(* Logix 5000 project; controller DispersionPlc vendor 1 type 14 code 108 rev 34.11; software revision 34.01; part 3 of 22 *)
(* tags used below, declared in another part *)
   Control_Rm_tags : DINT;
   Dev : REAL[10];
   DevAlarms : DINT;
   DevTimer : TIMER[10];
   Dispersion_to_Main : DINT;
   Dispersion_to_Main2 : DINT;
   Dispersion_to_SIL2 : DINT;
   Dispersion_to_SIL2_Analog : REAL[24];
   GenPurp : AStd_GeneralPurp;
   PLCStatus : AStd_PLCStatus;
   SP : REAL;

   T4301_AIR_PURGE : ALIAS FOR Local:6:O.Data.4;
   T4301_AIR_PURGE_AUTO : BOOL := 1;
   T4301_AIR_PURGE_REQUEST : BOOL;
   T4301_COOLING_NOT_PURGED : BOOL;
   T4301_COOLING_OCCURED : BOOL;
   T4301_Cooling_On : BOOL;
   T4301_COOLING_OPERATION : BOOL;
   T4301_Cooling_Reset_TMR : TIMER := (PRE := 500);
   T4301_COOLING_TEMP : DINT := 72;
   T4301_COOLING_VALVE : ALIAS FOR Local:6:O.Data.3;
   T4301_COOLING_VALVE_HMI : BOOL;
   T4301_DISCHARGE : BOOL;
   T4301_DISCHARGE_VALVE : AB:1769_DI16:I:0;
   T4301_Heating_On : BOOL;
   T4301_HEATING_OPERATION : BOOL;
   T4301_HMI_Cooling : BOOL;
   T4301_HMI_Heating : BOOL;
   T4301_K : Kettle := (Heating.Value := 78.0, Heating.Setpoint := 100.0, Heating.Error_Val := 115.0, Heating.OUT := 10000.0, Cooling.Value := 78.0, Cooling.Setpoint := 85.0, Cooling.Error_Val := 72.0, Cooling.OUT := 10000.0, Combined.Value := 78.0, Auto_Manual := 1, Cool_Auto_Manual := 1);
   T4301_Manual_AIR_PURGE_REQUEST : BOOL;
   T4301_Mixer : VFD := (TargetDriveSpeed := 100, I_CmdDir := 1, I_ActDir := 1, I_LocalContStat1 := 1, I_LocalContStat2 := 1, I_LocalContStat3 := 1, O_Stop := 1, O_DirBit1 := 1, O_Reff_Sel1 := 1, O_V_CmdReff := 11000.0, SpeedScaleIn := 110.0, SpeedScaleOut := 110.0, MaxOutPut := 100.0, MinOutput := 10.0);
   T4301_Mixer_Enable : DINT;
   T4301_PID_Setpoints : PID[5] := ([1].SP := 100.0, [1].KP := 325.0, [1].KI := 0.02, [2].KP := 9.0, [2].KI := 8.0, [2].KD := 7.0, [3].KP := 8.0, [3].KI := 0.2, [4].KP := 6.0, [4].KI := 5.0, [4].KD := 4.0);
   T4301_Pids_On : BOOL;
   T4301_Post_PurgeTm : DINT := 20000;
   T4301_Pre_PurgeTm : DINT := 2000;
   T4301_PrePurgeTMR : TIMER := (PRE := 2000);
   T4301_Process_Alarm_Setpoints : Alarm_SPT := (HIHI := 340.0, HI := 320.0);
   T4301_Purge_Complete : BOOL := 1;
   T4301_Request_Cooling : BOOL;
   T4301_Request_Cooling_Tmr : TIMER[5] := ([0].PRE := 30000, [1].PRE := 30000, [2].PRE := 500, [3].PRE := 8000, [4].PRE := 500, [4].ACC := 515, [4].EN := 1, [4].DN := 1);
   T4301_Request_Cooling_Tmr1 : TIMER := (PRE := 1000);
   T4301_Request_Heating : BOOL;
   T4301_Request_Heating_Hold : BOOL;
   T4301_Request_Heating_Tmr : TIMER[5] := ([0].PRE := 5000, [4].PRE := 5000, [4].ACC := 5006);
   T4301_Stop_Pids : BOOL;
   T4301_T4302_Xfer_In_Enable_Ctrl : BOOL := 1;
   T4301_Temp_Feed_Alarm : DINT := 310;
   T4301_Z1_HEAT_VALVE : ALIAS FOR Local:6:O.Data.0;
   T4301_Z2_HEAT_VALVE : ALIAS FOR Local:6:O.Data.1;
   T4301_Z3_HEAT_VALVE : ALIAS FOR Local:6:O.Data.2;
   T4301ons2 : DINT := 386;
   T4301PID_I : REAL;
   T4301Purge : Seq64 := (Val := 1, Tmr[3].PRE := 4000, Tmr[5].PRE := 20000, Sq.Step[1] := 1);
   T4302_AIR_PURGE : ALIAS FOR Local:6:O.Data.13;
   T4302_AIR_PURGE_AUTO : BOOL := 1;
   T4302_AIR_PURGE_REQUEST : BOOL;
   T4302_Cooling_No_Heat : TIMER := (PRE := 200000);
   T4302_COOLING_NOT_PURGED : BOOL;
   T4302_COOLING_OCCURED : BOOL;
   T4302_Cooling_On : BOOL := 1;
   T4302_COOLING_OPERATION : BOOL := 1;
   T4302_Cooling_Pressure : DINT;
   T4302_Cooling_Pressure_SPT : DINT := 50;
   T4302_COOLING_TEMP : DINT := 2192;
   T4302_COOLING_VALVE : ALIAS FOR Local:6:O.Data.10;
   T4302_COOLING_VALVE_HMI : BOOL;
   T4302_DISCHARGE : BOOL;
   T4302_Heating_On : BOOL;
   T4302_HEATING_OPERATION : BOOL;
   T4302_HMI_Cooling : BOOL;
   T4302_HMI_Heating : BOOL;
   T4302_K : Kettle := (Heating.Value := 65.0, Heating.Setpoint := 150.0, Heating.Error_Val := 95.0, Heating.OUT := 5000.0, Cooling.Value := 65.0, Cooling.Setpoint := 180.0, Combined.Value := 65.0, Combined.Setpoint := 287.0, Auto_Manual := 1, ValveOutput := 2, Cool_Auto_Manual := 1);
   t4302_Line_pressure_High : BOOL;
   t4302_Line_pressure_Hightmr : TIMER := (PRE := 20000);
   T4302_Manual_AIR_PURGE_REQUEST : BOOL;
   T4302_Mixer : VFD := (TargetDriveSpeed := 100, I_DatalinkA2_Fb := 223.0, O_DirBit1 := 1, O_Reff_Sel1 := 1, O_V_CmdReff := 11000.0, SpeedScaleIn := 110.0, SpeedScaleOut := 110.0, MaxOutPut := 100.0, MinOutput := 10.0);
   T4302_Phase_S52_Transfer : AStd_PLI := (IdleS := 1, CurrentStateCodeS := 1, PreventStartS := 2, AlarmS := 2, StepNo := 1, StepBit := 2, PreventStartInhibitC := 3, AlarmInhibitC := 3, IntSafDisp := 2);
   T4302_Phase_S52_Transfer_AOI : AStd_PLI_AOI := (PreventStartS := 1, AlmS := 1, StepNo := 1, cfgAutoReset := 1);
   T4302_Phase_TT_Transfer : AStd_PLI := (IdleS := 1, CurrentStateCodeS := 1, PreventStartS := 2, AlarmS := 2, StepNo := 1, StepBit := 2, RealParameters[0] := 44000.0, PreventStartInhibitC := 7, AlarmInhibitC := 3, IntSafDisp := 2);
   T4302_Phase_TT_Transfer_AOI : AStd_PLI_AOI := (PreventStartS := 1, AlmS := 1, StepNo := 1, cfgAutoReset := 1);
   T4302_PhaseAgitation : AStd_PLI := (IdleS := 1, CurrentStateCodeS := 1, StepNo := 1, StepBit := 2, DINTParameters[0] := 32, DINTParameters[1] := 8500, PreventStartInhibitC := 3, AlarmInhibitC := 3);
   T4302_PhaseAgitation_AOI : AStd_PLI_AOI := (StepNo := 1, cfgAutoReset := 1);
   T4302_PhaseTempControl : AStd_PLI := (IdleS := 1, CurrentStateCodeS := 1, StepNo := 1, StepBit := 2, RealParameters[0] := 65.0, RealParameters[1] := 64.0, RealParameters[3] := 50.0, RealParameters[4] := 113.0, RealParameters[5] := 50.0, RealParameters[10] := 5000.0, RealParameters[19] := 70.0, DINTParameters[0] := 5, DINTParameters[19] := 80, PreventStartInhibitC := 15, AlarmInhibitC := 15);
   T4302_PhaseTempControl_AOI : AStd_PLI_AOI := (StepNo := 1, cfgAutoReset := 1);
   T4302_PID_Setpoints : PID[5] := ([1].SP := 5.0, [1].KP := 150.0, [1].KI := 0.01, [2].KP := 9.0, [2].KI := 8.0, [2].KD := 7.0, [3].SP := 100.0, [3].KP := 8.0, [3].KI := 0.2, [4].KP := 6.0, [4].KI := 5.0, [4].KD := 4.0);
   T4302_Pids_On : BOOL := 1;
   T4302_Post_PurgeTm : DINT := 20000;
   T4302_Pre_PurgeTm : DINT := 2000;
   T4302_PrePurgeTMR : TIMER := (PRE := 2000);
   T4302_Process_Alarm_Setpoints : Alarm_SPT := (HIHI := 340.0, HI := 320.0);
   T4302_Purge_Complete : BOOL := 1;
   T4302_RampControl : BOOL;
   T4302_RampControl_ONS : BOOL;
   T4302_RampControl_ONS_2 : BOOL;
   T4302_RampControlTOn : TIMER := (PRE := 600000);
   T4302_Request_Cooling : BOOL;
   T4302_Request_Cooling_Tmr : TIMER[5] := ([0].PRE := 20000, [1].PRE := 20000, [2].PRE := 500, [3].PRE := 8000, [4].PRE := 500, [4].ACC := 506, [4].EN := 1, [4].DN := 1);
   T4302_Request_Heating : BOOL;
   T4302_Request_Heating_Hold : BOOL;
   T4302_Request_Heating_Tmr : TIMER[5] := ([0].PRE := 1000, [4].PRE := 1000, [4].ACC := 1000);
   T4302_Stop_Pids : BOOL;
   T4302_Temp_Feed_Alarm : DINT := 310;
   T4302_TransferStarted : BOOL;
   T4302_Z1_HEAT_VALVE : ALIAS FOR Local:6:O.Data.9;
   T4302_Z2_HEAT_VALVE : ALIAS FOR Local:6:O.Data.8;
   T4302_Z3_HEAT_VALVE : ALIAS FOR Local:6:O.Data.11;
   T4302ons2 : DINT := 258;
   T4302Ons3 : BOOL := 1;
   T4302ons4 : BOOL;
   T4302Purge : Seq64 := (Val := 1, Tmr[3].PRE := 4000, Tmr[5].PRE := 2000, Sq.Step[1] := 1);
   T4302TruckTransferCompletePB : BOOL;
   T430_Z3_HEAT_VALVE : ALIAS FOR Local:6:O.Data.11;
   T47_Amount_Per_Count : REAL;
   T47_Charge_Remaining : REAL;
   T47_Flow_Rate : REAL;
   T47_Flow_Raw : DINT;
   T47_Flow_Raw_Adjusted : REAL;
   T47_Flow_Scale_Factor : REAL;
   T47_Last_Charge : REAL;
   T47_Manual_Start : BOOL;
   T47_Max_Flow : REAL;
   T47_Pump_Manual_Run : BOOL;
   T47_Pump_Off : BOOL;
   T47_Pump_Run : BOOL;
   T47_Transfer : BOOL;
   T47_transfer_amount : REAL;
   T47PumpTmr : TIMER;
   T51_Tank_Max_Lbs : REAL := 75000.0;
   T52_Mixer : VFD := (TargetDriveSpeed := 30, I_Ready := 1, I_CmdDir := 1, I_ActDir := 1, I_LocalContStat1 := 1, I_LocalContStat2 := 1, I_LocalContStat3 := 1, O_V_CmdReff := 4530.0, SpeedScaleIn := 151.0, SpeedScaleOut := 151.0, MaxOutPut := 100.0, MinOutput := 10.0);
   T52_Mixer_STOP : TIMER := (PRE := 200, ACC := 202, EN := 1, DN := 1);
   T52_Ons : BOOL[32] := ([20] := 1);
   T52_Selected_For_Pumping : BOOL;
   T52_Tank_Max_Lbs : REAL := 108286.0;
   T52_WARN_BYPASS : BOOL;
   T53_Mixer : VFD := (TargetDriveSpeed := 30, I_Ready := 1, I_CmdDir := 1, I_ActDir := 1, I_LocalContStat1 := 1, I_LocalContStat2 := 1, I_LocalContStat3 := 1, O_V_CmdReff := 4530.0, SpeedScaleIn := 151.0, SpeedScaleOut := 151.0, MaxOutPut := 100.0, MinOutput := 10.0);
   T53_Mixer_STOP : TIMER := (PRE := 200, ACC := 201, EN := 1, DN := 1);
   T53_Ons : BOOL[32];
   T53_Selected_For_Pumping : BOOL := 1;
   T53_Tank_Max_Lbs : REAL := 108286.0;
   T53_WARN_BYPASS : BOOL;
   T_4301_Temp_Holding : REAL := 78.06781;
   T_4301_Temp_Samples : REAL := 1000.0;
   T_4302_Temp_Holding : REAL := 66.95962;
   T_4302_Temp_Samples : REAL := 1000.0;
   T_4302_Temp_Smoothed : REAL := 66.95962;
   TA_4303 : ALIAS FOR Local:7:O.Data.13;
   TAH_4304 : ALIAS FOR Local:7:O.Data.12;
   Tank : Udt_Tank[64];
   tank1 : DINT;
   Tank47_Level : INT;
   Tank47_LevelHiHiAlarm : BOOL;
   Tank_Destination : DINT;
   Tank_Destination_ONS : BOOL;
   Tank_Destination_ONS1 : BOOL;
   Tank_Link_Enable : BOOL := 1;
   Tank_Link_Enable_ONS : BOOL;
   Tank_Link_Enable_ONS1 : BOOL;
   Tank_Link_ONS : BOOL[32];
   Tank_Linked : BOOL := 1;
   Task_OLD_Permissive : BOOL[64];
   Task_Permissive : DINT[2] := ([0] := 4, [1] := 4);
   TC_4305_1 : AStd_PIDInterface := (AutoS := 1, SPC := 65.0, PGainC := 1.0, IGainC := 0.33, DGainC := 0.22, PGainS := 1.0, IGainS := 0.33, DGainS := 0.22, SPS := 65.0, PVS := 76.673004, Perm.IntlkS := 1, Perm.SafeS := 1);
   TC_4305_1_AOI : AStd_PIDInterface_AOI := (SP := 65.0, PV := 76.642, cfgPVMaxEU := 350.0);
   TC_4305_1_PID : PID_ENHANCED := (PV := 76.673004, PVEUMax := 350.0, SPProg := 65.0, SPOper := 65.0, SPHLimit := 350.0, RatioProg := 1.0, RatioOper := 1.0, RatioHLimit := 1.0, RatioLLimit := 1.0, CVEUMax := 100.0, CVHLimit := 100.0, DependIndepend := 1, PGain := 1.0, IGain := 0.33, DGain := 0.22, PVHHLimit := 350.0, PVHLimit := 350.0, PVLLimit := 0.1, PVLLLimit := 0.1, DevHHLimit := 5.0, DevDeadband := 2.0, ProgProgReq := 1, ProgOverrideReq := 1, RTSTime := 1, SP := 65.0, SPPercent := 18.571428, PVPercent := 21.906572, E := -11.673004, EPercent := -3.335144, InitPrimary := 1, Ratio := 1.0, DevHHAlarm := 1, ProgOper := 1, Override := 1, DeltaT := 0.1);
   TCV_4302_1 : AStd_VlvModulating := (AutoC := 1, AutoS := 1, Perm.IntlkS := 1, Perm.SafeS := 1, Perm.InterlockInhibitC := 3, Scaling.RawMaxS := 10000.0, Scaling.EngMaxS := 100.0);
   TCV_4302_1_AOI : AStd_VlVModulating_AOI := (cfgEUMax := 100.0, cfgRawMax := 10000.0, AutoS := 1);
   TCV_4302_2 : AStd_VlvModulating := (AutoC := 1, AutoS := 1, Perm.IntlkS := 1, Perm.SafeS := 1, AutoPosC[0] := 100.0, AutoPosS := 100.0, Scaling.RawMaxS := 10000.0, Scaling.EngMaxS := 100.0);
   TCV_4302_2_AOI : AStd_VlVModulating_AOI := (cfgEUMax := 100.0, cfgRawMax := 10000.0, AutoS := 1);
   TCV_4302_2_Mode : SINT := 1;
   TCV_4305_1 : AStd_VlvModulating := (AutoC := 1, AutoS := 1, Perm.IntlkS := 1, Perm.SafeS := 1, Perm.InterlockInhibitC := 3, Perm.SafetyInhibitC := 255, Scaling.RawMaxS := 10000.0, Scaling.EngMaxS := 100.0);
   TCV_4305_1_AOI : AStd_VlVModulating_AOI := (cfgEUMax := 100.0, cfgRawMax := 10000.0, AutoS := 1);
   TCV_S47_1 : AStd_AnalogInput := (Raw := 4000.0, Scaled := 644000.0, Scaling.RawMaxS := 100.0, Scaling.EngMinS := 4000.0, Scaling.EngMaxS := 20000.0, High.LatchA := 1, High.DetectS := 1, High.BitS := 1, High.Tmr.PRE := 1000, High.Tmr.ACC := 1003, High.Tmr.EN := 1, High.Tmr.DN := 1, HighHigh.LatchA := 1, HighHigh.DetectS := 1, HighHigh.BitS := 1, HighHigh.Tmr.PRE := 1000, HighHigh.Tmr.ACC := 1003, HighHigh.Tmr.EN := 1, HighHigh.Tmr.DN := 1);
   TCV_S47_1_AOI : AStd_AI_AOI := (InputRaw_I := 4000.0, cfgRawMax := 100.0, cfgEUMin := 4000.0, cfgEUMax := 20000.0, Scaled := 644000.0);
   TCV_S47_1_AutoCommand : REAL;
   TCV_S47_1_AutoManTransition : BOOL;
   TCV_S47_1_AutoManTransitionDelay : TIMER := (PRE := 500);
   TCV_S47_1_AutoPB : BOOL;
   TCV_S47_1_AutoSelected : BOOL;
   TCV_S47_1_Command : REAL;
   TCV_S47_1_ManAutoTransition : BOOL;
   TCV_S47_1_ManAutoTransitionDelay : TIMER := (PRE := 500);
   TCV_S47_1_ManualCommand : DINT;
   TCV_S47_1_ManualPB : BOOL;
   TCV_S47_1_ManualSelected : BOOL;
   TCV_S47_1Output : Analog_Scale := (Analog_Max_In := 100.0, Analog_Min_Out := 4000.0, Analog_Max_Out := 20000.0, Analog_Out := 4000.0);
   TE_4301A : ALIAS FOR Local:8:I.Ch0Data;
   Te_4301A_High : REAL := 420.0;
   TE_4301A_Low : REAL := 20.0;
   Te_4301A_max : REAL;
   TE_4301B : ALIAS FOR Local:8:I.Ch1Data;
   TE_4301C : REAL;
   TE_4301D : ALIAS FOR Local:8:I.Ch3Data;
   TE_4301E : ALIAS FOR Local:8:I.Ch4Data;
   TE_4302A : ALIAS FOR Local:8:I.Ch5Data;
   TE_4302A_High : REAL := 420.0;
   TE_4302A_Low : REAL := 20.0;
   TE_4302B : REAL;
   TE_4302C : ALIAS FOR Local:8:I.Ch2Data;
   TE_4302D : REAL;
   TE_4302E : REAL;
   TE_4303 : ALIAS FOR Local:9:I.Ch4Data;
   TE_4303_01 : REAL := 66.38342;
   TE_4303_High : REAL := 90.0;
   TE_4304 : ALIAS FOR Local:9:I.Ch5Data;
   TE_4304_High : REAL := 95.0;
   TE_4320 : INT := 143;
   TE_4320_High : REAL := 160.0;
   TE_4320_Raw : DINT;
   TE_K400_1 : REAL := 5.0;
   TE_K400_1_HIGH : REAL := 300.0;
   TE_K400_1_LOW : REAL := 50.0;
   TempChange : REAL := 54.0;
   TempDifferenceCooling4301 : DINT := 14;
   TempDifferenceCooling4301TMR : TIMER := (PRE := 600000);
   TempDifferenceCooling4302 : DINT := -115;
   TempDifferenceCooling4302TMR : TIMER := (PRE := 600000);
   test1 : BOOL;
   test3 : BOOL;
   TEST_1 : INT;
   TEST_2 : BOOL;
   test_618 : BOOL := 1;
   TEST_INTERLOCK_K400 : BOOL;
   TEST_INTERLOCK_RESET : DINT;
   TEST_INTERLOCK_T4301 : BOOL;
   TEST_INTERLOCK_T4302 : BOOL;
   test_onsite_512 : BOOL;
   test_onsite_514 : BOOL;
   Test_PID : PID_ENHANCED := (PVEUMax := 100.0, SPHLimit := 100.0, RatioProg := 1.0, RatioOper := 1.0, RatioHLimit := 1.0, RatioLLimit := 1.0, CVEUMax := 100.0, CVHLimit := 100.0, PVEDerivative := 1, RTSTime := 1, InitPrimary := 1, Ratio := 1.0, Manual := 1, DeltaT := 0.1);
   TestBit1 : BOOL;
   TestBit2 : BOOL;
   TestBit3 : BOOL := 1;
   testint : DINT;
   testons : DINT;
   testtmr : TIMER[5] := ([0].PRE := 500, [1].PRE := 500, [1].ACC := 500, [1].EN := 1, [1].DN := 1);
   tete : BOOL;
   tg : BOOL;
   THINONS1 : BOOL;
   THO_MSG : MESSAGE;
        MessageParameters(ServiceCode := 16#0fa2, LocalElement := TO_N12[0], ...)
   THRM_OX_ALM_AUX : ALIAS FOR Local:1:I.Data[1].17;
   TIC_4302_1 : AStd_PIDInterface := (AutoS := 1, SPC := 167.0, PGainC := 5.0, IGainC := 0.1, DGainC := 0.5, PGainS := 5.0, IGainS := 0.1, DGainS := 0.5, SPS := 167.0, PVS := 75.0, Perm.IntlkS := 1, Perm.SafeS := 1);
   TIC_4302_1_AOI : AStd_PIDInterface_AOI := (SP := 167.0, PV := 75.0, cfgPVMaxEU := 400.0);
   TIC_4302_1_PID : PID_ENHANCED := (PV := 75.0, PVEUMax := 400.0, SPProg := 167.0, SPOper := 167.0, SPHLimit := 400.0, RatioProg := 1.0, RatioOper := 1.0, RatioHLimit := 1.0, RatioLLimit := 1.0, CVEUMax := 225.0, CVEUMin := 70.0, CVHLimit := 100.0, PGain := 5.0, IGain := 0.1, DGain := 0.5, PVEDerivative := 1, DevDeadband := 2.0, ProgProgReq := 1, ProgOverrideReq := 1, RTSTime := 1, CVEU := 70.0, SP := 167.0, SPPercent := 41.75, PVPercent := 18.75, E := 92.0, EPercent := 23.0, InitPrimary := 1, Ratio := 1.0, ProgOper := 1, Override := 1, DeltaT := 0.1);
   TIC_4302_4C : AStd_PIDInterface := (AutoS := 1, SPC := 65.0, PGainC := 3.9, IGainC := 0.28, DGainC := 0.125, PGainS := 3.9, IGainS := 0.28, DGainS := 0.125, SPS := 65.0, PVS := 75.991, Perm.IntlkS := 1, Perm.SafeS := 1);
   TIC_4302_4C_AOI : AStd_PIDInterface_AOI := (SP := 65.0, PV := 76.022, cfgPVMinEU := 40.0, cfgPVMaxEU := 350.0);
   TIC_4302_4C_PID : PID_ENHANCED := (PV := 76.022, PVEUMax := 350.0, PVEUMin := 40.0, SPProg := 65.0, SPOper := 65.0, SPHLimit := 350.0, SPLLimit := 40.0, RatioProg := 1.0, RatioOper := 1.0, RatioHLimit := 1.0, RatioLLimit := 1.0, CVEUMax := 100.0, CVHLimit := 100.0, ControlAction := 1, DependIndepend := 1, PGain := 3.9, IGain := 0.28, DGain := 0.125, DevDeadband := 2.0, ProgProgReq := 1, ProgOverrideReq := 1, RTSTime := 1, SP := 65.0, SPPercent := 8.064516, PVPercent := 11.609999, E := 10.990997, EPercent := 3.5454826, InitPrimary := 1, Ratio := 1.0, ProgOper := 1, Override := 1, DeltaT := 0.1);
   TIC_4302_4H : AStd_PIDInterface := (AutoS := 1, SPC := 65.0, PGainC := 4.8, IGainC := 0.31, DGainC := 0.19, PGainS := 4.8, IGainS := 0.31, DGainS := 0.19, SPS := 65.0, PVS := 76.022, Perm.IntlkS := 1, Perm.SafeS := 1);
   TIC_4302_4H_AOI : AStd_PIDInterface_AOI := (SP := 65.0, PV := 76.022, cfgPVMinEU := 40.0, cfgPVMaxEU := 350.0);
   TIC_4302_4H_PID : PID_ENHANCED := (PV := 76.022, PVEUMax := 350.0, PVEUMin := 40.0, SPProg := 65.0, SPOper := 65.0, SPHLimit := 350.0, SPLLimit := 40.0, RatioProg := 1.0, RatioOper := 1.0, RatioHLimit := 1.0, RatioLLimit := 1.0, CVEUMax := 100.0, CVHLimit := 80.0, DependIndepend := 1, PGain := 4.8, IGain := 0.31, DGain := 0.19, DevDeadband := 2.0, ProgProgReq := 1, ProgOverrideReq := 1, RTSTime := 1, SP := 65.0, SPPercent := 8.064516, PVPercent := 11.620001, E := -11.022003, EPercent := -3.5554848, InitPrimary := 1, Ratio := 1.0, ProgOper := 1, Override := 1, DeltaT := 0.1);
   TIC_4302_4H_PID_01 : PID_ENHANCED := (PVEUMax := 100.0, SPHLimit := 100.0, RatioProg := 1.0, RatioOper := 1.0, RatioHLimit := 1.0, RatioLLimit := 1.0, CVEUMax := 100.0, CVHLimit := 100.0, PVEDerivative := 1, RTSTime := 1);
   TIT_4302_1 : AStd_AnalogInput := (Raw := 75.0, Scaled := 75.0, Scaling.RawMinS := 60.0, Scaling.RawMaxS := 500.0, Scaling.EngMinS := 60.0, Scaling.EngMaxS := 500.0, LowLow.LimitC := 25.0, LowLow.Tmr.PRE := 1000, LowLow.Disabled := 1, Low.LimitC := 50.0, Low.Tmr.PRE := 1000, Low.Disabled := 1, High.LimitC := 350.0, High.Tmr.PRE := 1000, High.Disabled := 1, HighHigh.LimitC := 375.0, HighHigh.Tmr.PRE := 1000, HighHigh.Disabled := 1, Fault.LimitC := 40.0, Fault.LimitOffSetC := 20.0, Fault.Tmr.PRE := 5000, FaultReset := 5.0);
   TIT_4302_1_AOI : AStd_AI_AOI := (InputRaw_I := 75.0, cfgRawMin := 60.0, cfgRawMax := 500.0, cfgEUMin := 60.0, cfgEUMax := 500.0, Scaled := 75.0);
   TIT_4302_1_sim_Val : DINT := 155;
   TIT_4302_1_Simulation : BOOL := 1;
   TIT_4302_4 : AStd_AnalogInput := (Raw := 1161.0, Scaled := 75.991, Scaling.RawMaxS := 10000.0, Scaling.EngMinS := 40.0, Scaling.EngMaxS := 350.0, LowLow.LimitC := 25.0, LowLow.Tmr.PRE := 60000, LowLow.Disabled := 1, Low.LimitC := 50.0, Low.LimitOffSetC := 5.0, Low.Tmr.PRE := 60000, High.LimitC := 250.0, High.LimitOffSetC := 5.0, High.Tmr.PRE := 60000, HighHigh.LimitC := 375.0, HighHigh.Tmr.PRE := 60000, HighHigh.Disabled := 1, Fault.LimitC := -1000.0, Fault.LimitOffSetC := 1000.0, Fault.Tmr.PRE := 10000, FaultReset := 500.0);
   TIT_4302_4_AOI : AStd_AI_AOI := (InputRaw_I := 1162.0, cfgRawMax := 10000.0, cfgEUMin := 40.0, cfgEUMax := 350.0, Scaled := 76.022);
   TIT_4302_4_sim_Val : DINT := 200;
   TIT_4302_4_Simulation : BOOL := 1;
   TIT_4302_5 : AStd_AnalogInput := (Raw := 1113.0, Scaled := 74.503, Scaling.RawMaxS := 10000.0, Scaling.EngMinS := 40.0, Scaling.EngMaxS := 350.0, LowLow.LimitC := 20.0, LowLow.Tmr.PRE := 5000, LowLow.Disabled := 1, Low.LimitC := 10.0, Low.Tmr.PRE := 1000, Low.Disabled := 1, High.LimitC := 350.0, High.Tmr.PRE := 1000, High.Disabled := 1, HighHigh.LimitC := 375.0, HighHigh.Tmr.PRE := 1000, HighHigh.Disabled := 1, Fault.LimitC := -1000.0, Fault.LimitOffSetC := 1000.0, Fault.Tmr.PRE := 10000, FaultReset := 500.0);
   TIT_4302_5_AOI : AStd_AI_AOI := (InputRaw_I := 1114.0, cfgRawMax := 10000.0, cfgEUMin := 40.0, cfgEUMax := 350.0, Scaled := 74.534);
   TIT_4305_1 : AStd_AnalogInput := (Raw := 1183.0, Scaled := 76.673004, Scaling.RawMaxS := 10000.0, Scaling.EngMinS := 40.0, Scaling.EngMaxS := 350.0, LowLow.LimitC := 40.0, LowLow.LimitOffSetC := 5.0, LowLow.Tmr.PRE := 60000, LowLow.Disabled := 1, Low.LimitC := 50.0, Low.LimitOffSetC := 20.0, Low.Tmr.PRE := 60000, Low.Disabled := 1, High.LimitC := 150.0, High.LimitOffSetC := 50.0, High.Tmr.PRE := 60000, High.Disabled := 1, HighHigh.LimitC := 190.0, HighHigh.LimitOffSetC := 5.0, HighHigh.Tmr.PRE := 60000, HighHigh.Disabled := 1, Fault.LimitC := -1000.0, Fault.LimitOffSetC := 1000.0, Fault.Tmr.PRE := 5000, FaultReset := 500.0);
   TIT_4305_1_AOI : AStd_AI_AOI := (InputRaw_I := 1182.0, cfgRawMax := 10000.0, cfgEUMin := 40.0, cfgEUMax := 350.0, Scaled := 76.642, CommsStatus := 1);
   TIT_4305_1_sim_Val : DINT := 200;
   TIT_4305_1_Simulation : BOOL := 1;
   TIT_4306_1 : AStd_AnalogInput := (Raw := 1251.0, Scaled := 72.526, Scaling.RawMaxS := 10000.0, Scaling.EngMinS := 40.0, Scaling.EngMaxS := 300.0, LowLow.LimitC := 100.0, LowLow.Tmr.PRE := 30000, LowLow.Disabled := 1, Low.LimitC := 85.0, Low.Tmr.PRE := 30000, Low.Disabled := 1, High.LimitC := 190.0, High.Tmr.PRE := 30000, High.Disabled := 1, HighHigh.LimitC := 200.0, HighHigh.Tmr.PRE := 30000, HighHigh.Disabled := 1, Fault.LimitC := -1000.0, Fault.LimitOffSetC := 1000.0, Fault.Tmr.PRE := 5000, FaultReset := 500.0);
   TIT_4306_1_AOI : AStd_AI_AOI := (InputRaw_I := 1252.0, cfgRawMax := 10000.0, cfgEUMin := 40.0, cfgEUMax := 300.0, Scaled := 72.552);
   TIT_4306_1_sim_Val : DINT := 189;
   TIT_4306_1_Simulation : BOOL := 1;
   TIT_4307_1 : AStd_AnalogInput := (Raw := 920.0, Scaled := 73.119995, Scaling.RawMaxS := 10000.0, Scaling.EngMinS := 40.0, Scaling.EngMaxS := 400.0, LowLow.LimitC := 90.0, LowLow.Tmr.PRE := 30000, LowLow.Disabled := 1, Low.LimitC := 85.0, Low.Tmr.PRE := 30000, Low.Disabled := 1, High.LimitC := 200.0, High.Tmr.PRE := 30000, High.Disabled := 1, HighHigh.LimitC := 140.0, HighHigh.Tmr.PRE := 30000, HighHigh.Disabled := 1, Fault.LimitC := -1000.0, Fault.LimitOffSetC := 1000.0, Fault.Tmr.PRE := 5000, FaultReset := 500.0);
   TIT_4307_1_AOI : AStd_AI_AOI := (InputRaw_I := 919.0, cfgRawMax := 10000.0, cfgEUMin := 40.0, cfgEUMax := 400.0, Scaled := 73.084);
   TIT_4307_1_sim_Val : DINT := 249;
   TIT_4307_1_Simulation : BOOL := 1;
   TIT_K200_2_AOI : AStd_AI_AOI := (InputRaw_I := 4526.0, cfgRawMin := -3460.0, cfgRawMax := 21920.0, cfgEUMax := 10.0, Scaled := 3.146572);
   TIT_K200_3 : AStd_AnalogInput := (Raw := 8048.0, Scaled := 156.38, Scaling.RawMinS := 4000.0, Scaling.RawMaxS := 20000.0, Scaling.EngMinS := 40.0, Scaling.EngMaxS := 500.0, LowLow.Disabled := 1, Low.LimitC := 50.0, Low.Tmr.PRE := 1000, Low.Disabled := 1, High.LimitC := 350.0, High.Disabled := 1, HighHigh.LimitC := 375.0, HighHigh.Tmr.PRE := 1000, Fault.LimitC := 4000.0, Fault.Tmr.PRE := 1000);
   TIT_K200_3_AOI : AStd_AI_AOI := (InputRaw_I := 8048.0, cfgRawMin := 4000.0, cfgRawMax := 20000.0, cfgEUMin := 40.0, cfgEUMax := 500.0, Scaled := 156.38);
   TIT_K200_3_Val : REAL := 8046.0;
   TIT_K400_1 : AStd_AnalogInput := (Raw := 319.7, Scaled := 319.7, Scaling.RawMaxS := 1000.0, Scaling.EngMaxS := 1000.0, LowLow.LimitC := 90.0, LowLow.Tmr.PRE := 1000, LowLow.Disabled := 1, Low.LatchA := 1, Low.DetectS := 1, Low.BitS := 1, Low.LimitC := 340.0, Low.Tmr.PRE := 1000, Low.Tmr.ACC := 1015, Low.Tmr.EN := 1, Low.Tmr.DN := 1, High.LimitC := 1700.0, High.Tmr.PRE := 1000, High.Disabled := 1, HighHigh.LimitC := 400.0, HighHigh.Tmr.PRE := 1000, HighHigh.Disabled := 1, Fault.LimitC := -10.0, Fault.LimitOffSetC := 10.0, Fault.Tmr.PRE := 1000, FaultReset := 5.0);
   TIT_K400_1_AOI : AStd_AI_AOI := (InputRaw_I := 319.80002, cfgRawMax := 1000.0, cfgEUMax := 1000.0, Scaled := 319.80002, CommsStatus := 1);
   TIT_K400_1_sim_Val : DINT := 25;
   TIT_K400_1_Simulation : BOOL := 1;
   TIT_K400_1_Val : REAL := 319.80002;
   TIT_K400_3 : AStd_AnalogInput := (Raw := -2500.0, Scaled := -50.0, Scaling.RawMaxS := 10000.0, Scaling.EngMinS := 60.0, Scaling.EngMaxS := 500.0, LowLow.LatchA := 1, LowLow.DetectS := 1, LowLow.BitS := 1, LowLow.LimitC := 195.0, LowLow.LimitOffSetC := 5.0, LowLow.Tmr.PRE := 30000, LowLow.Tmr.ACC := 30010, LowLow.Tmr.EN := 1, LowLow.Tmr.DN := 1, Low.LimitC := 50.0, Low.Tmr.PRE := 30000, Low.Disabled := 1, High.LimitC := 350.0, High.Tmr.PRE := 30000, High.Disabled := 1, HighHigh.LimitC := 375.0, HighHigh.Tmr.PRE := 30000, HighHigh.Disabled := 1, Fault.LatchA := 1, Fault.DetectS := 1, Fault.BitS := 1, Fault.Tmr.PRE := 5000, Fault.Tmr.ACC := 5003, Fault.Tmr.EN := 1, Fault.Tmr.DN := 1);
   TIT_K400_3_AOI : AStd_AI_AOI := (InputRaw_I := -2500.0, cfgRawMax := 10000.0, cfgEUMin := 60.0, cfgEUMax := 500.0, Scaled := -50.0);
   TIT_K400_3_sim_Val : DINT := 250;
   TIT_K400_3_Simulation : BOOL;
   TIT_S47_1 : AStd_AnalogInput := (Raw := 6749.0, Scaled := 68.1075, Scaling.RawMinS := 4000.0, Scaling.RawMaxS := 20000.0, Scaling.EngMinS := 20.0, Scaling.EngMaxS := 300.0, LowLow.Tmr.PRE := 1000, Low.Tmr.PRE := 1000, High.LatchA := 1, High.DetectS := 1, High.BitS := 1, High.Tmr.PRE := 1000, High.Tmr.ACC := 1007, High.Tmr.EN := 1, High.Tmr.DN := 1, HighHigh.LatchA := 1, HighHigh.DetectS := 1, HighHigh.BitS := 1, HighHigh.Tmr.PRE := 1000, HighHigh.Tmr.ACC := 1007, HighHigh.Tmr.EN := 1, HighHigh.Tmr.DN := 1, Fault.LimitC := 4000.0, Fault.Tmr.PRE := 1000);
   TIT_S47_1_AOI : AStd_AI_AOI := (InputRaw_I := 6749.0, cfgRawMin := 4000.0, cfgRawMax := 20000.0, cfgEUMin := 20.0, cfgEUMax := 300.0, Scaled := 68.1075);
   TIT_S47_1_HiHi : REAL := 150.0;
   TIT_S51_1 : AStd_AnalogInput := (Raw := 14392.0, Scaled := 162.375, Scaling.RawMinS := 4000.0, Scaling.RawMaxS := 20000.0, Scaling.EngMaxS := 250.0, LowLow.LimitC := 80.0, LowLow.LimitOffSetC := 5.0, LowLow.Tmr.PRE := 300000, Low.LimitC := -100.0, Low.LimitOffSetC := 5.0, Low.Tmr.PRE := 300000, High.LimitC := 350.0, High.Tmr.PRE := 300000, High.Disabled := 1, HighHigh.LimitC := 375.0, HighHigh.Tmr.PRE := 300000, HighHigh.Disabled := 1, Fault.LimitC := 4000.0, Fault.Tmr.PRE := 5000);
   TIT_S51_1_AOI : AStd_AI_AOI := (InputRaw_I := 14397.0, cfgRawMin := 4000.0, cfgRawMax := 20000.0, cfgEUMax := 250.0, Scaled := 162.45312, CommsStatus := 1);
   TIT_S51_1_Raw : DINT := 14396;
   TIT_S51_2 : AStd_AnalogInput;
   TIT_S51_3 : AStd_AnalogInput;
   tm3 : TIMER := (PRE := 300000);
   tmrtest : BOOL;
   TO_Alarm : BOOL;
   TO_Alarm_Int : INT := 2;
   TO_ALARM_MSG_DINT : DINT := 2;
   To_CtrlRm1 : MESSAGE;
        MessageParameters(ServiceCode := 16#004c, LocalElement := Control_Rm_tags, ...)
   To_CtrlRm2 : MESSAGE;
        MessageParameters(ServiceCode := 16#004c, LocalElement := TIT_K400_1_Val, ...)
   To_CtrlRm3 : MESSAGE;
        MessageParameters(ServiceCode := 16#004c, LocalElement := TT_K200_2_Raw, ...)
   To_Dispersion_PLC : DINT;
   To_Main : MESSAGE;
        MessageParameters(ServiceCode := 16#004d, LocalElement := Dispersion_to_Main, ...)
   To_Main2 : MESSAGE;
        MessageParameters(ServiceCode := 16#004d, LocalElement := Dispersion_to_Main2, ...)
   TO_Message : MESSAGE;
        MessageParameters(ServiceCode := 16#0fa2, LocalElement := TO_N12[0], ...)
   TO_N12 : INT[100] := ([0] := 1254, [1] := 70, [2] := 1525, [3] := 625, [4] := 725, [7] := 1525, [8] := 100, [9] := 626, [10] := 728, [11] := 3, [12] := -20, [13] := 20, [14] := 37, [15] := 60, [16] := 61, [17] := 21, [18] := 21, [20] := 1000, [21] := 20, [22] := 27, [24] := 800, [26] := 1, [27] := 1, [33] := 12, [36] := 1, [37] := 45, [38] := 3073, [39] := 300, [41] := 45, [43] := 35, [44] := 495, [45] := 35, [46] := 2, [47] := 1000, [49] := 72, [50] := 20, [52] := 100, [54] := 100, [59] := 480, [60] := -5);
   To_SIL2 : MESSAGE;
        MessageParameters(ServiceCode := 16#004d, LocalElement := Dispersion_to_SIL2, ...)
   To_SIL2_Analog : MESSAGE;
        MessageParameters(ServiceCode := 16#004d, LocalElement := Dispersion_to_SIL2_Analog[0], ...)
   TO_SIL2_PLC : DINT[3];
   tog1 : BOOL := 1;
   TOGGLE : BOOL;
   TOGGLE1 : BOOL := 1;
   ToMesTmr : TIMER := (PRE := 1000, ACC := 398, EN := 1, TT := 1);
   TR_4320_Open : ALIAS FOR Local:1:I.Data[8].8;
   Trans_Pump_P52_Aux : ALIAS FOR Local:1:I.Data[33].0;
   Trans_Pump_P53_Aux : ALIAS FOR Local:1:I.Data[33].1;
   TRANS_PUMP_P_4301_AUX : ALIAS FOR Local:1:I.Data[1].1;
   TRANS_PUMP_P_4301_RUN : ALIAS FOR Local:1:O.Data[0].1;
   TRANS_PUMP_P_4302_AUX : ALIAS FOR Local:1:I.Data[1].3;
   TRANS_PUMP_P_4302_RUN : ALIAS FOR Local:1:O.Data[0].3;
   TRANS_PUMP_P_4320_AUX : ALIAS FOR Local:1:I.Data[1].6;
   TRANS_PUMP_P_4320_RUN : ALIAS FOR Local:1:O.Data[0].6;
   Trans_Pump_T52_Run : ALIAS FOR Local:1:O.Data[13].1;
   Trans_Pump_T52_Run_Lamp : ALIAS FOR Local:1:O.Data[12].0;
   Trans_Pump_T52_Run_LampA : ALIAS FOR Local:1:O.Data[22].0;
   Trans_Pump_T52_Run_PB : ALIAS FOR Local:1:I.Data[27].0;
   Trans_Pump_T52_RunA : ALIAS FOR Local:1:O.Data[23].1;
   Trans_Pump_T52_Stop_PB : ALIAS FOR Local:1:I.Data[27].1;
   Trans_Pump_T53_Run : ALIAS FOR Local:1:O.Data[13].2;
   Trans_Pump_T53_Run_Lamp : ALIAS FOR Local:1:O.Data[12].1;
   Trans_Pump_T53_Run_LampA : ALIAS FOR Local:1:O.Data[12].1;
   Trans_Pump_T53_Run_LampB : ALIAS FOR Local:1:O.Data[22].1;
   Trans_Pump_T53_Run_PB : ALIAS FOR Local:1:I.Data[27].2;
   Trans_Pump_T53_RunA : ALIAS FOR Local:1:O.Data[13].2;
   Trans_Pump_T53_RunB : ALIAS FOR Local:1:O.Data[23].2;
   Trans_Pump_T53_Stop_PB : ALIAS FOR Local:1:I.Data[27].3;
   TransferDone : BOOL;
   TransferOffset : REAL := 100.0;
   TransferSetpoint : REAL := 44000.0;
   TransferStopValueLb : REAL := 43900.0;
   TruckLoadLevelAlarmHIHI : BOOL;
   TruckLoadLevelAlarmHIHIRedundant : BOOL;
   TruckLoadLevelAlarmResetPB : BOOL;
   TruckLoadLevelAlarmResetPBLight : BOOL := 1;
   TT_K200_2 : REAL := 480.9;
   TT_K200_2_Raw : DINT := 4809;
   V4304_Pump : VFD := (TargetDriveSpeed := 64, I_Ready := 1, I_Running := 1, I_CmdDir := 1, I_ActDir := 1, I_AtSpeed := 1, I_LocalContStat1 := 1, I_LocalContStat2 := 1, I_LocalContStat3 := 1, I_Act_Amps := 1.0, O_Run := 1, O_DirBit1 := 1, O_Reff_Sel1 := 1, O_V_CmdReff := 9728.0, SpeedScaleIn := 151.25, SpeedScaleOut := 152.0, MaxOutPut := 100.0, MinOutput := 10.0, DriveSpeedReff := 64.31735);
   V4304_Pump_TargetDriveSpeed_Timer : TIMER := (PRE := 30000);
   V4306_Barcode : STRING[8] := ([0] := '75380', [1] := '75381', [2] := '75382');
   V4306_PhaseAddRO : AStd_PLI := (IdleS := 1, CurrentStateCodeS := 1, StepNo := 1, StepBit := 2);
   V4306_PhaseAddRO_AOI : AStd_PLI_AOI := (StepNo := 1, cfgAutoReset := 1);
   V4306_PhaseAgitation : AStd_PLI := (IdleS := 1, CurrentStateCodeS := 1, StepNo := 1, StepBit := 2, DINTParameters[0] := 55, DINTParameters[1] := 250, DINTParameters[18] := 30, DINTParameters[19] := 5, PreventStartInhibitC := 15, AlarmInhibitC := 15);
   V4306_PhaseAgitation_AOI : AStd_PLI_AOI := (StepNo := 1, cfgAutoReset := 1);
   V4306_PhaseHeat : AStd_PLI := (IdleS := 1, CurrentStateCodeS := 1, StepNo := 1, StepBit := 2, RealParameters[0] := 106.0, RealParameters[10] := 250.0, RealParameters[11] := 107.0, RealParameters[12] := 10.0, RealParameters[13] := 5.0, RealParameters[14] := 3.0, RealParameters[15] := 5.0, RealParameters[16] := 195.0, RealParameters[17] := 200.0, RealParameters[18] := 208.0, RealParameters[19] := 210.0, PreventStartInhibitC := 253, AlarmInhibitC := 255);
   V4306_PhaseHeat_AOI : AStd_PLI_AOI := (StepNo := 1, cfgAutoReset := 1);
   V4306_PhaseRunPumpCirculate : AStd_PLI := (IdleS := 1, CurrentStateCodeS := 1, StepNo := 1, StepBit := 2, PreventStartInhibitC := 15, AlarmInhibitC := 7, InterlockTimers.Timers[0].PRE := 10000, InterlockTimers.Timers[1].PRE := 5000);
   V4306_PhaseRunPumpCirculate_AOI : AStd_PLI_AOI := (StepNo := 1, cfgAutoReset := 1);
   V4306_PhaseRunPumpDrumAdd : AStd_PLI := (IdleS := 1, CurrentStateCodeS := 1, StepNo := 1, StepBit := 2, RealParameters[0] := -1.0, RealParameters[1] := 175.6, PreventStartInhibitC := 15, AlarmInhibitC := 23, InterlockTimers.Timers[0].PRE := 10000, InterlockTimers.Timers[1].PRE := 5000);
   V4306_PhaseRunPumpDrumAdd_AOI : AStd_PLI_AOI := (StepNo := 1, cfgAutoReset := 1);
   V4306_PhaseRunPumpDrumAddCompleteC : BOOL;
   V4306_PhaseTransfer : AStd_PLI := (IdleS := 1, CurrentStateCodeS := 1, StepNo := 1, StepBit := 2, RealParameters[0] := 51.199997, RealParameters[1] := 59.0, RealParameters[2] := 2.199997, RealParameters[3] := 53.641064, RealParameters[4] := 50.799995, RealParameters[5] := 1.77, RealParameters[6] := 59.0, RealParameters[7] := 1.0, RealParameters[8] := 10.0, RealParameters[19] := 0.03, PreventStartInhibitC := 204, AlarmInhibitC := 204);
   V4306_PhaseTransfer_AOI : AStd_PLI_AOI := (StepNo := 1, cfgAutoReset := 1);
   V4306_PhaseTransfer_DelayTimer : TIMER := (PRE := 1000);
   V4306_Scan_Read_Delay : TIMER := (PRE := 1000);
   V4306_Transfer_LineClear : TIMER := (PRE := 10000);
   V4307_PhaseAddRO : AStd_PLI := (IdleS := 1, CurrentStateCodeS := 1, StepNo := 1, StepBit := 2, UnitProc_PhaseID := 1111);
   V4307_PhaseAddRO_AOI : AStd_PLI_AOI := (StepNo := 1, cfgPhaseID := 1111);
   V4307_PhaseAgitation : AStd_PLI := (IdleS := 1, CurrentStateCodeS := 1, StepNo := 1, StepBit := 2, DINTParameters[0] := 50, DINTParameters[1] := 325);
   V4307_PhaseAgitation_AOI : AStd_PLI_AOI := (StepNo := 1, cfgAutoReset := 1);
   V4307_PhaseCool : AStd_PLI := (IdleS := 1, CurrentStateCodeS := 1, StepNo := 1, StepBit := 2, UnitProc_PhaseID := 1111, RealParameters[0] := 105.0, RealParameters[10] := 325.0, RealParameters[11] := 104.0, RealParameters[12] := 5.0, RealParameters[13] := 3.0, RealParameters[14] := 5.0, RealParameters[15] := 10.0, RealParameters[16] := 245.0, RealParameters[17] := 247.0, RealParameters[18] := 255.0, RealParameters[19] := 260.0, PreventStartInhibitC := 254, AlarmInhibitC := 252);
   V4307_PhaseCool_AOI : AStd_PLI_AOI := (StepNo := 1, cfgAutoReset := 1, cfgPhaseID := 1111);
   V4307_PhaseRunPumpCirculate : AStd_PLI := (IdleS := 1, CurrentStateCodeS := 1, StepNo := 1, StepBit := 2, PreventStartInhibitC := 31, AlarmInhibitC := 7);
   V4307_PhaseRunPumpCirculate_AOI : AStd_PLI_AOI := (StepNo := 1, cfgAutoReset := 1);
   V4307_PhaseTransfer : AStd_PLI := (IdleS := 1, CurrentStateCodeS := 1, StepNo := 1, StepBit := 2, UnitProc_PhaseID := 1111, RealParameters[0] := 82.94, RealParameters[1] := 89.0, RealParameters[2] := 3.9400024, RealParameters[3] := 84.24333, RealParameters[4] := 80.86, RealParameters[5] := 2.6699998, RealParameters[6] := 89.0, RealParameters[7] := 1.0, RealParameters[8] := 10.0, RealParameters[19] := 0.03, PreventStartInhibitC := 124, AlarmInhibitC := 12);
   V4307_PhaseTransfer_AOI : AStd_PLI_AOI := (StepNo := 1, cfgAutoReset := 1, cfgPhaseID := 1111);
   V4307_PhaseTransfer_DelayTimer : TIMER := (PRE := 1000);
   V4307_Transfer_LineClear : TIMER := (PRE := 10000);
   Vaild_Monomer_Barcode : BOOL;
   Vaild_Monomer_Barcode_At_Index : DINT;
   Vaild_Monomer_BarcodeS : STRING[20] := ([0] := '813142859744', [1] := '813143559744', [2] := '813202859744', [3] := '813202859733', [4] := '821137758207', [5] := '821137759733', [6] := '821137754404', [7] := '821137758231', [8] := '821224158207', [9] := '821224154404', [10] := '813142810313', [11] := '813143558106', [12] := '813202858106', [13] := '821137758116', [14] := '821224159504', [15] := '710844125998', [16] := '710844158059');
   VFD_4302_1 : AStd_VFD := (AutoS := 1, ManSpdC := 32.0, AutoSpdS := 32.0, SpeedI.Scaling.RawMaxS := 60.0, SpeedI.Scaling.EngMaxS := 100.0, SpeedC.Scaling.RawMaxS := 60.0, SpeedC.Scaling.EngMaxS := 100.0, DiscI := 1, RunTimeS := 10017, Perm.IntlkS := 1, Perm.SafeS := 1, Perm.InterlockInhibitC := 3, Perm.SafetyInhibitC := 3, MiscAlm.Tmr.PRE := 20000, DiscAlm.Tmr.PRE := 10000);
   VFD_4302_1_AOI : AStd_VFD_AOI := (DirectionFWD_O := 1, AutoS := 1, cfgHasRunFdbk := 1, cfgHasSpeedFdbk := 1, cfgRawMax := 60.0, cfgEUMax := 100.0);
   VFD_4302_1_Simulation : BOOL := 1;
   VFD_4306_1 : AStd_VFD := (AutoS := 1, ManSpdC := 55.0, AutoSpdS := 55.0, SpeedI.Scaling.RawMaxS := 6000.0, SpeedI.Scaling.EngMaxS := 100.0, SpeedI.LowLow.LimitC := 5.0, SpeedI.LowLow.LimitOffSetC := 5.0, SpeedI.Low.LimitC := 10.0, SpeedI.Low.LimitOffSetC := 5.0, SpeedI.High.LimitC := 70.0, SpeedI.High.LimitOffSetC := 5.0, SpeedI.HighHigh.LimitC := 90.0, SpeedI.HighHigh.LimitOffSetC := 5.0, SpeedC.Scaling.RawMaxS := 6000.0, SpeedC.Scaling.EngMaxS := 100.0, DiscI := 1, RunTimeS := 1045, Perm.IntlkS := 1, Perm.SafeS := 1, Perm.InterlockInhibitC := 1, Perm.InterlockTimers.Timers[0].PRE := 5000, MiscAlm.Tmr.PRE := 20000, DiscAlm.Tmr.PRE := 5000);
   VFD_4306_1_AOI : AStd_VFD_AOI := (DirectionFWD_O := 1, AutoS := 1, cfgHasRunFdbk := 1, cfgHasSpeedFdbk := 1, cfgRawMax := 6000.0, cfgEUMax := 100.0);
   VFD_4306_1_Simulation : BOOL := 1;
   VFD_4307_1 : AStd_VFD := (AutoS := 1, ManSpdC := 20.0, AutoSpdS := 50.0, SpeedI.Scaling.RawMaxS := 6000.0, SpeedI.Scaling.EngMaxS := 100.0, SpeedC.Scaling.RawMaxS := 6000.0, SpeedC.Scaling.EngMaxS := 100.0, DiscI := 1, RunTimeS := 1694, Perm.IntlkS := 1, Perm.SafeS := 1, Perm.InterlockInhibitC := 1, Perm.SafetyInhibitC := 1, MiscAlm.Tmr.PRE := 20000, DiscAlm.Tmr.PRE := 5000);
   VFD_4307_1_AOI : AStd_VFD_AOI := (DirectionFWD_O := 1, AutoS := 1, cfgHasRunFdbk := 1, cfgHasSpeedFdbk := 1, cfgRawMax := 6000.0, cfgEUMax := 100.0);
   VFD_4307_1_Simulation : BOOL := 1;
   VFD_P_4302_2 : AStd_VFD := (AutoS := 1, ManSpdC := 80.0, AutoSpdS := 80.0, SpeedI.Scaling.RawMaxS := 6000.0, SpeedI.Scaling.EngMaxS := 100.0, SpeedC.Scaling.RawMaxS := 6000.0, SpeedC.Scaling.EngMaxS := 100.0, DiscI := 1, RunTimeS := 10435, Perm.IntlkS := 1, Perm.SafeS := 1, Perm.InterlockInhibitC := 1, Perm.SafetyInhibitC := 1, MiscAlm.Tmr.PRE := 20000, DiscAlm.Tmr.PRE := 10000);
   VFD_P_4302_2_AOI : AStd_VFD_AOI := (DirectionFWD_O := 1, AutoS := 1, cfgHasRunFdbk := 1, cfgHasSpeedFdbk := 1, cfgRawMax := 6000.0, cfgEUMax := 100.0);
   VFD_P_4302_2_Simulation : BOOL := 1;
   W2_High_Level : BOOL;
   W2_W4_High_Level : BOOL;
   W4303_Pump : VFD := (TargetDriveSpeed := 86, I_Ready := 1, I_Running := 1, I_CmdDir := 1, I_ActDir := 1, I_AtSpeed := 1, I_LocalContStat1 := 1, I_LocalContStat2 := 1, I_LocalContStat3 := 1, I_Act_Amps := 2.0, O_Run := 1, O_DirBit1 := 1, O_Reff_Sel1 := 1, O_V_CmdReff := 8600.0, SpeedScaleIn := 100.0, SpeedScaleOut := 100.0, MaxOutPut := 100.0, MinOutput := 10.0, DriveSpeedReff := 86.0);
   W4_High_Level : BOOL;
   WallClockCurrent : DINT[2] := ([0] := 1990006213, [1] := 230852);
   WallClockDiff : DINT[2] := ([0] := 17153);
   WallClockPrevious : DINT[2] := ([0] := 1990126269, [1] := 230852);
   WI_4310 : REAL := 843.2;
   WI_4310_OffSet : REAL;
   WI_4310_Sf : REAL;
   WIT_4302_1 : AStd_AnalogInput := (Raw := 3917.285, Scaled := 946.56824, Scaling.RawMinS := 4000.0, Scaling.RawMaxS := 20000.0, Scaling.EngMinS := 1240.0, Scaling.EngMaxS := 58000.0, LowLow.LimitC := 2000.0, LowLow.Tmr.PRE := 60000, LowLow.Disabled := 1, Low.LimitC := 3000.0, Low.Tmr.PRE := 60000, Low.Disabled := 1, High.LimitC := 47000.0, High.LimitOffSetC := 1000.0, High.Tmr.PRE := 60000, HighHigh.LimitC := 48000.0, HighHigh.LimitOffSetC := 2000.0, HighHigh.Tmr.PRE := 60000, Fault.LimitC := 3000.0, Fault.LimitOffSetC := 1000.0, Fault.Tmr.PRE := 5000, FaultReset := 500.0);
   WIT_4302_1_AOI : AStd_AI_AOI := (InputRaw_I := 3917.5334, cfgRawMin := 4000.0, cfgRawMax := 20000.0, cfgEUMin := 1240.0, cfgEUMax := 58000.0, Scaled := 947.44995, CommsStatus := 1);
   WIT_4302_1_HH : TIMER := (PRE := 5000);
   WIT_4302_1_sim_Val : DINT := 20000;
   WIT_4302_1_Simulation : BOOL := 1;
   WIT_4306_1 : AStd_AnalogInput := (Raw := 9.0, Scaled := 1.8, Scaling.RawMaxS := 10000.0, Scaling.EngMaxS := 2000.0, LowLow.LimitC := 100.0, LowLow.LimitOffSetC := 10.0, LowLow.Tmr.PRE := 10000, LowLow.Disabled := 1, Low.LimitC := 200.0, Low.LimitOffSetC := 10.0, Low.Tmr.PRE := 10000, Low.Disabled := 1, High.LimitC := 1600.0, High.LimitOffSetC := 100.0, High.Tmr.PRE := 10000, HighHigh.LimitC := 1700.0, HighHigh.LimitOffSetC := 100.0, HighHigh.Tmr.PRE := 10000, Fault.LimitC := -1000.0, Fault.LimitOffSetC := 1000.0, Fault.Tmr.PRE := 5000, FaultReset := 500.0);
   WIT_4306_1_AOI : AStd_AI_AOI := (InputRaw_I := 8.0, cfgRawMax := 10000.0, cfgEUMax := 2000.0, Scaled := 1.5999999, CommsStatus := 1);
   WIT_4306_1_sim_Val : REAL := 800.0;
   WIT_4306_1_Simulation : BOOL := 1;
   WIT_4307_1 : AStd_AnalogInput := (Raw := 1.0, Scaled := 0.26, Scaling.RawMaxS := 10000.0, Scaling.EngMaxS := 2600.0, LowLow.LimitC := 200.0, LowLow.LimitOffSetC := 10.0, LowLow.Tmr.PRE := 10000, LowLow.Disabled := 1, Low.LimitC := 400.0, Low.LimitOffSetC := 10.0, Low.Tmr.PRE := 10000, Low.Disabled := 1, High.LimitC := 2300.0, High.LimitOffSetC := 100.0, High.Tmr.PRE := 10000, HighHigh.LimitC := 2400.0, HighHigh.LimitOffSetC := 100.0, HighHigh.Tmr.PRE := 10000, Fault.LimitC := -1000.0, Fault.LimitOffSetC := 1000.0, Fault.Tmr.PRE := 5000, FaultReset := 500.0);
   WIT_4307_1_AOI : AStd_AI_AOI := (InputRaw_I := 1.0, cfgRawMax := 10000.0, cfgEUMax := 2600.0, Scaled := 0.26, CommsStatus := 1);
   WIT_4307_1_sim_Val : DINT := 900;
   WIT_4307_1_Simulation : BOOL := 1;
   XI_K400_1 : BOOL := 1;
   XV_3001 : ALIAS FOR Local:5:O.Data.10;
   XV_4301 : ALIAS FOR Local:5:O.Data.0;
   XV_4301_01_PB : BOOL;
   XV_4301_1 : AStd_VlvOC := (CloseO := 1, ClosedI := 1, cfgHasZSC := 1, CycleCountS := 16, Perm.IntlkS := 1, Perm.SafeS := 1, Perm.InterlockInhibitC := 3, MiscAlm.InhibitC := 1, MiscAlm.Tmr.PRE := 30000);
   XV_4301_1_AOI : AStd_VlvOC_AOI := (Closed_I := 1, Close_O := 1, cfgHasZSC := 1);
   XV_4301_1_IOpn : BOOL;
   XV_4301_1_OCls : BOOL := 1;
   XV_4301_1_OOpn : BOOL;
   XV_4301_8 : AStd_VlvOC := (AutoS := 1, CloseO := 1, ClosedI := 1, cfgHasZSC := 1, CycleCountS := 360, Perm.IntlkS := 1, Perm.SafeS := 1, Perm.InterlockInhibitC := 127, Perm.SafetyInhibitC := 127, MiscAlm.Tmr.PRE := 30000);
   XV_4301_8_AOI : AStd_VlvOC_AOI := (AutoS := 1, Closed_I := 1, Close_O := 1, cfgHasZSC := 1);
   XV_4301_8_IOpn : BOOL;
   XV_4301_8_OCls : BOOL := 1;
   XV_4301_8_Simulation : BOOL := 1;
   XV_4302 : ALIAS FOR Local:5:O.Data.1;
   XV_4302_1 : AStd_VlvOC := (CloseO := 1, ClosedI := 1, cfgHasZSC := 1, CycleCountS := 39, Perm.IntlkS := 1, Perm.SafeS := 1, MiscAlm.InhibitC := 1, MiscAlm.Tmr.PRE := 30000);
   XV_4302_10 : AStd_VlvOC := (AutoS := 1, CloseO := 1, ClosedI := 1, cfgHasZSC := 1, CycleCountS := 1589, Perm.IntlkS := 1, Perm.SafeS := 1, Perm.InterlockInhibitC := 63, Perm.SafetyInhibitC := 63, Perm.InterlockTimers.Timers[5].PRE := 30000, MiscAlm.Tmr.PRE := 30000);
   XV_4302_10_AOI : AStd_VlvOC_AOI := (AutoS := 1, Closed_I := 1, Close_O := 1, cfgHasZSC := 1);
   XV_4302_10_IOpn : BOOL;
   XV_4302_10_OCls : BOOL := 1;
   XV_4302_10_Simulation : BOOL;
   XV_4302_11 : AStd_VlvOC := (CloseO := 1, ClosedI := 1, cfgHasZSC := 1, CycleCountS := 24, Perm.IntlkS := 1, Perm.SafeS := 1, Perm.InterlockInhibitC := 3, Perm.IntSafDisp := 4, MiscAlm.Tmr.PRE := 30000);
   XV_4302_11_AOI : AStd_VlvOC_AOI := (Closed_I := 1, Close_O := 1, cfgHasZSC := 1);
   XV_4302_11_IOpn : BOOL;
   XV_4302_11_OCls : BOOL := 1;
   XV_4302_11_OOpn : BOOL;
   XV_4302_11Sol : BOOL;
   XV_4302_12 : AStd_VlvOC := (CloseO := 1, ClosedI := 1, cfgHasZSC := 1, cfgHasZSO := 1, CycleCountS := 103, Perm.IntlkS := 1, Perm.SafeS := 1, MiscAlm.Tmr.PRE := 30000);
   XV_4302_12_AOI : AStd_VlvOC_AOI := (Closed_I := 1, Close_O := 1, cfgHasZSO := 1, cfgHasZSC := 1);
   XV_4302_12_ClosedI : ALIAS FOR Local:4:I.Data.2;
   XV_4302_12_IOpn : BOOL;
   XV_4302_12_OCls : BOOL := 1;
   XV_4302_12_OpenI : ALIAS FOR Local:4:I.Data.3;
   XV_4302_12_OpenO : ALIAS FOR Local:6:O.Data.5;
   XV_4302_13 : AStd_VlvOC := (AutoS := 1, CloseO := 1, ClosedI := 1, cfgHasZSC := 1, cfgHasZSO := 1, CycleCountS := 41, Perm.IntlkS := 1, Perm.SafeS := 1, Perm.InterlockInhibitC := 1, Perm.SafetyInhibitC := 1, Perm.IntSafDisp := 1, MiscAlm.Tmr.PRE := 30000);
   XV_4302_13_AOI : AStd_VlvOC_AOI := (AutoS := 1, Closed_I := 1, Close_O := 1, cfgHasZSO := 1, cfgHasZSC := 1); {access Read Only}
   XV_4302_13_ClosedI : ALIAS FOR Local:1:I.Data[27].23;
   XV_4302_13_IOpn : BOOL; {access Read Only}
   XV_4302_13_OCls : BOOL := 1; {access Read Only}
   XV_4302_13_OpenC : ALIAS FOR Local:1:O.Data[12].17;
   XV_4302_13_OpenI : ALIAS FOR Local:1:I.Data[27].24;
   XV_4302_1_AOI : AStd_VlvOC_AOI := (Closed_I := 1, Close_O := 1, cfgHasZSC := 1);
   XV_4302_1_IOpn : BOOL;
   XV_4302_1_OCls : BOOL := 1;
   XV_4302_1_OOpn : BOOL;
   XV_4302_2 : AStd_VlvOC := (CloseO := 1, AlmS := 1, cfgHasZSC := 1, Perm.IntlkS := 1, Perm.SafeS := 1, MiscAlm.LatchA := 1, MiscAlm.DetectS := 1, MiscAlm.BitS := 1, MiscAlm.Tmr.PRE := 30000, MiscAlm.Tmr.ACC := 30007, MiscAlm.Tmr.EN := 1, MiscAlm.Tmr.DN := 1);
   XV_4302_2_AOI : AStd_VlvOC_AOI := (AlmS := 1, Close_O := 1, cfgHasZSC := 1);
   XV_4302_2_ICls : BOOL;
   XV_4302_2_IOpn : BOOL;
   XV_4302_2_OCls : BOOL := 1;
   XV_4302_2_OOpn : BOOL;
   XV_4302_2_Simulation : BOOL;
   XV_4302_3 : AStd_VlvOC := (CloseO := 1, AlmS := 1, cfgHasZSC := 1, Perm.IntlkS := 1, Perm.SafeS := 1, MiscAlm.LatchA := 1, MiscAlm.DetectS := 1, MiscAlm.BitS := 1, MiscAlm.Tmr.PRE := 30000, MiscAlm.Tmr.ACC := 30007, MiscAlm.Tmr.EN := 1, MiscAlm.Tmr.DN := 1);
   XV_4302_3_AOI : AStd_VlvOC_AOI := (AlmS := 1, Close_O := 1, cfgHasZSC := 1);
   XV_4302_3_ICls : BOOL;
   XV_4302_3_IOpn : BOOL;
   XV_4302_3_OCls : BOOL := 1;
   XV_4302_3_OOpn : BOOL;
   XV_4302_3_Simulation : BOOL;
   XV_4302_4 : AStd_VlvOC := (CloseO := 1, AlmS := 1, cfgHasZSC := 1, Perm.IntlkS := 1, Perm.SafeS := 1, MiscAlm.LatchA := 1, MiscAlm.DetectS := 1, MiscAlm.BitS := 1, MiscAlm.Tmr.PRE := 30000, MiscAlm.Tmr.ACC := 30007, MiscAlm.Tmr.EN := 1, MiscAlm.Tmr.DN := 1);
   XV_4302_4_AOI : AStd_VlvOC_AOI := (AlmS := 1, Close_O := 1, cfgHasZSC := 1);
   XV_4302_4_ICls : BOOL;
   XV_4302_4_IOpn : BOOL;
   XV_4302_4_OCls : BOOL := 1;
   XV_4302_4_OOpn : BOOL;
   XV_4302_4_Simulation : BOOL;
   XV_4302_5 : AStd_VlvOC := (AutoS := 1, CloseO := 1, ClosedI := 1, cfgHasZSC := 1, CycleCountS := 535, Perm.IntlkS := 1, Perm.SafeS := 1, Perm.InterlockInhibitC := 3, Perm.SafetyInhibitC := 3, MiscAlm.Tmr.PRE := 30000);
   XV_4302_5_AOI : AStd_VlvOC_AOI := (AutoS := 1, Closed_I := 1, Close_O := 1, cfgHasZSC := 1);
   XV_4302_5_IOpn : BOOL;
   XV_4302_5_OCls : BOOL := 1;
   XV_4302_5_Simulation : BOOL;
   XV_4302_6 : AStd_VlvOC := (AutoS := 1, CloseO := 1, ClosedI := 1, cfgHasZSC := 1, CycleCountS := 65, Perm.IntlkS := 1, Perm.SafeS := 1, MiscAlm.Tmr.PRE := 30000);
   XV_4302_6_AOI : AStd_VlvOC_AOI := (AutoS := 1, Closed_I := 1, Close_O := 1, cfgHasZSC := 1);
   XV_4302_6_IOpn : BOOL;
   XV_4302_6_OCls : BOOL := 1;
   XV_4302_6_Simulation : BOOL;
   XV_4302_7 : AStd_VlvOC := (AutoS := 1, CloseO := 1, ClosedI := 1, cfgHasZSC := 1, CycleCountS := 23, Perm.IntlkS := 1, Perm.SafeS := 1, Perm.InterlockInhibitC := 1, Perm.SafetyInhibitC := 1, MiscAlm.Tmr.PRE := 30000);
   XV_4302_7_AOI : AStd_VlvOC_AOI := (AutoS := 1, Closed_I := 1, Close_O := 1, cfgHasZSC := 1);
   XV_4302_7_IOpn : BOOL;
   XV_4302_7_OCls : BOOL := 1;
   XV_4302_7_Simulation : BOOL;
   XV_4302_8 : AStd_VlvOC := (AutoS := 1, CloseO := 1, ClosedI := 1, cfgHasZSC := 1, CycleCountS := 946, Perm.IntlkS := 1, Perm.SafeS := 1, Perm.InterlockInhibitC := 511, Perm.SafetyInhibitC := 511, MiscAlm.Tmr.PRE := 30000);
   XV_4302_8_AOI : AStd_VlvOC_AOI := (AutoS := 1, Closed_I := 1, Close_O := 1, cfgHasZSC := 1);
   XV_4302_8_IOpn : BOOL;
   XV_4302_8_OCls : BOOL := 1;
   XV_4302_8_Simulation : BOOL;
   XV_4302_9 : AStd_VlvOC := (AutoS := 1, CloseO := 1, ClosedI := 1, cfgHasZSC := 1, CycleCountS := 63, Perm.IntlkS := 1, Perm.SafeS := 1, Perm.InterlockInhibitC := 1, MiscAlm.Tmr.PRE := 30000);
   XV_4302_9_AOI : AStd_VlvOC_AOI := (AutoS := 1, Closed_I := 1, Close_O := 1, cfgHasZSC := 1);
   XV_4302_9_IOpn : BOOL;
   XV_4302_9_OCls : BOOL := 1;
   XV_4302_9_Simulation : BOOL := 1;
   XV_4303_01 : ALIAS FOR Local:5:O.Data.3;
   XV_4303_01_PB : BOOL;
   XV_4303_02 : ALIAS FOR Local:7:O.Data.8;
   XV_4303_02_ZSC : BOOL := 1;
   XV_4303_02_ZSO : BOOL;
   XV_4303_03 : BOOL;
   XV_4303_03_Enable : DINT := 1;
   XV_4303_04 : BOOL;
   XV_4303_05 : BOOL := 1;
   XV_4304 : ALIAS FOR Local:5:O.Data.4;
   XV_4304_02 : BOOL;
   XV_4304_02_Enable : DINT := 1;
   XV_4304_03 : BOOL;
   XV_4304_04 : BOOL := 1;
   XV_4306_1 : AStd_VlvOC := (AutoS := 1, CloseO := 1, ClosedI := 1, cfgHasZSC := 1, CycleCountS := 1148, Perm.IntlkS := 1, Perm.SafeS := 1, MiscAlm.Tmr.PRE := 30000);
   XV_4306_1_AOI : AStd_VlvOC_AOI := (AutoS := 1, Closed_I := 1, Close_O := 1, cfgHasZSC := 1);
   XV_4306_1_IOpn : BOOL;
   XV_4306_1_OCls : BOOL := 1;
   XV_4306_1_Simulation : BOOL;
   XV_4306_2 : AStd_VlvOC := (AutoS := 1, CloseO := 1, ClosedI := 1, cfgHasZSC := 1, CycleCountS := 475, Perm.IntlkS := 1, Perm.SafeS := 1, MiscAlm.Tmr.PRE := 30000);
   XV_4306_2_AOI : AStd_VlvOC_AOI := (AutoS := 1, Closed_I := 1, Close_O := 1, cfgHasZSC := 1);
   XV_4306_2_IOpn : BOOL;
   XV_4306_2_OCls : BOOL := 1;
   XV_4306_2_Simulation : BOOL;
   XV_4306_3 : AStd_VlvOC := (AutoS := 1, CloseO := 1, ClosedI := 1, cfgHasZSC := 1, CycleCountS := 643, Perm.IntlkS := 1, Perm.SafeS := 1, Perm.InterlockInhibitC := 511, Perm.SafetyInhibitC := 511, Perm.InterlockTimers.Timers[0].PRE := 10000, Perm.InterlockTimers.Timers[1].PRE := 4000, Perm.InterlockTimers.Timers[2].PRE := 60000, Perm.InterlockTimers.Timers[3].PRE := 60000, Perm.InterlockTimers.Timers[4].PRE := 5000, Perm.InterlockTimers.Timers[5].PRE := 30000, Perm.InterlockTimers.Timers[6].PRE := 30000, Perm.InterlockTimers.Timers[7].PRE := 30000, MiscAlm.Tmr.PRE := 30000);
   XV_4306_3_AOI : AStd_VlvOC_AOI := (AutoS := 1, Closed_I := 1, Close_O := 1, cfgHasZSC := 1);
   XV_4306_3_IOpn : BOOL;
   XV_4306_3_OCls : BOOL := 1;
   XV_4306_3_Simulation : BOOL;
   XV_4306_4 : AStd_VlvOC := (AutoS := 1, CloseO := 1, ClosedI := 1, cfgHasZSC := 1, CycleCountS := 680, Perm.IntlkS := 1, Perm.SafeS := 1, MiscAlm.Tmr.PRE := 30000);
   XV_4306_4_AOI : AStd_VlvOC_AOI := (AutoS := 1, Closed_I := 1, Close_O := 1, cfgHasZSC := 1);
   XV_4306_4_IOpn : BOOL;
   XV_4306_4_OCls : BOOL := 1;
   XV_4306_4_Simulation : BOOL;
   XV_4306_5 : AStd_VlvOC := (AutoS := 1, CloseO := 1, ClosedI := 1, cfgHasZSC := 1, CycleCountS := 1092, Perm.IntlkS := 1, Perm.SafeS := 1, Perm.InterlockInhibitC := 7, Perm.SafetyInhibitC := 7, Perm.InterlockTimers.Timers[0].PRE := 5000, Perm.InterlockTimers.Timers[1].PRE := 5000, Perm.InterlockTimers.Timers[2].PRE := 30000, MiscAlm.Tmr.PRE := 30000);
   XV_4306_5_AOI : AStd_VlvOC_AOI := (AutoS := 1, Closed_I := 1, Close_O := 1, cfgHasZSC := 1);
   XV_4306_5_IOpn : BOOL;
   XV_4306_5_OCls : BOOL := 1;
   XV_4306_5_Simulation : BOOL;
   XV_4307_1 : AStd_VlvOC := (AutoS := 1, CloseO := 1, ClosedI := 1, cfgHasZSC := 1, CycleCountS := 379, Perm.IntlkS := 1, Perm.SafeS := 1, MiscAlm.Tmr.PRE := 30000);
   XV_4307_1_AOI : AStd_VlvOC_AOI := (AutoS := 1, Closed_I := 1, Close_O := 1, cfgHasZSC := 1);
   XV_4307_1_IOpn : BOOL;
   XV_4307_1_OCls : BOOL := 1;
   XV_4307_1_Simulation : BOOL;
   XV_4307_2 : AStd_VlvOC := (AutoS := 1, CloseO := 1, ClosedI := 1, cfgHasZSC := 1, CycleCountS := 111, Perm.IntlkS := 1, Perm.SafeS := 1, MiscAlm.Tmr.PRE := 30000);
   XV_4307_2_AOI : AStd_VlvOC_AOI := (AutoS := 1, Closed_I := 1, Close_O := 1, cfgHasZSC := 1);
   XV_4307_2_IOpn : BOOL;
   XV_4307_2_OCls : BOOL := 1;
   XV_4307_2_Simulation : BOOL;
   XV_4307_3 : AStd_VlvOC := (AutoS := 1, CloseO := 1, ClosedI := 1, cfgHasZSC := 1, CycleCountS := 598, Perm.IntlkS := 1, Perm.SafeS := 1, Perm.InterlockInhibitC := 511, Perm.SafetyInhibitC := 511, Perm.InterlockTimers.Timers[7].PRE := 30000, MiscAlm.Tmr.PRE := 30000);
   XV_4307_3_AOI : AStd_VlvOC_AOI := (AutoS := 1, Closed_I := 1, Close_O := 1, cfgHasZSC := 1);
   XV_4307_3_IOpn : BOOL;
   XV_4307_3_OCls : BOOL := 1;
   XV_4307_3_Simulation : BOOL;
   XV_4307_4 : AStd_VlvOC := (AutoS := 1, CloseO := 1, ClosedI := 1, cfgHasZSC := 1, CycleCountS := 112, Perm.IntlkS := 1, Perm.SafeS := 1, MiscAlm.Tmr.PRE := 30000);
   XV_4307_4_AOI : AStd_VlvOC_AOI := (AutoS := 1, Closed_I := 1, Close_O := 1, cfgHasZSC := 1);
   XV_4307_4_IOpn : BOOL;
   XV_4307_4_OCls : BOOL := 1;
   XV_4307_4_Simulation : BOOL;
   XV_4307_6 : AStd_VlvOC := (AutoS := 1, CloseO := 1, ClosedI := 1, cfgHasZSC := 1, CycleCountS := 433, Perm.IntlkS := 1, Perm.SafeS := 1, Perm.InterlockInhibitC := 7, Perm.SafetyInhibitC := 7, Perm.InterlockTimers.Timers[0].PRE := 5000, Perm.InterlockTimers.Timers[2].PRE := 30000, MiscAlm.Tmr.PRE := 30000);
   XV_4307_6_AOI : AStd_VlvOC_AOI := (AutoS := 1, Closed_I := 1, Close_O := 1, cfgHasZSC := 1);
   XV_4307_6_IOpn : BOOL;
   XV_4307_6_OCls : BOOL := 1;
   XV_4307_6_Simulation : BOOL;
   XV_4320_1 : ALIAS FOR Local:1:O.Data[1].1;
   XV_4320_2 : ALIAS FOR Local:1:O.Data[1].0;
   XV_5201 : ALIAS FOR Local:1:O.Data[12].8;
   XV_5201A : ALIAS FOR Local:1:O.Data[22].8;
   XV_5202 : ALIAS FOR Local:1:O.Data[12].9;
   XV_5202A : ALIAS FOR Local:1:O.Data[22].9;
   XV_5301 : ALIAS FOR Local:1:O.Data[12].6;
   XV_5301A : ALIAS FOR Local:1:O.Data[22].6;
   XV_5302 : ALIAS FOR Local:1:O.Data[12].7;
   XV_5302A : ALIAS FOR Local:1:O.Data[22].7;
   XV_ISOLATION_VALVE : BOOL := 1;
   XV_K400_03_SEQCLOSE : BOOL;
   XV_K400_03_SEQOPEN : BOOL;
   XV_K400_04_SEQCLOSE : BOOL;
   XV_K400_04_SEQOPEN : BOOL;
   XV_K400_6 : AStd_VlvOC := (OpenO := 1, OpenI := 1, cfgHasZSC := 1, CycleCountS := 123, Perm.IntlkS := 1, Perm.SafeS := 1, Perm.InterlockInhibitC := 1, Perm.SafetyInhibitC := 1, MiscAlm.Tmr.PRE := 30000);
   XV_K400_6_AOI : AStd_VlvOC_AOI := (OpenS := 1, Open_O := 1, cfgHasZSC := 1);
   XV_K400_6_IOpn : BOOL;
   XV_K400_6_OCls : BOOL;
   XV_K400_6_Simulation : BOOL := 1;
   XV_K400_7 : AStd_VlvOC := (AutoS := 1, CloseO := 1, ClosedI := 1, cfgHasZSC := 1, CycleCountS := 34, Perm.InterlockS := 1, Perm.SafetyS := 1, Perm.InterlockInhibitC := 1, Perm.SafetyInhibitC := 1, Perm.IntSafDisp := 1, MiscAlm.Tmr.PRE := 30000);
   XV_K400_7_AOI : AStd_VlvOC_AOI := (AutoS := 1, Closed_I := 1, Close_O := 1, cfgHasZSC := 1);
   XV_K400_7_IOpn : BOOL;
   XV_K400_7_OCls : BOOL := 1;
   XV_K400_7_Simulation : BOOL := 1;
   XV_S47_1 : AStd_VlvOC;
   XV_S47_1_AOI : AStd_VlvOC_AOI := (cfgHasZSO := 1);
   XV_S47_1_CloseCommand : BOOL;
   XV_S47_1_IOpn : BOOL;
   XV_S47_1_IsClosed : BOOL := 1;
   XV_S47_1_IsOpen : BOOL;
   XV_S47_1_OCls : BOOL;
   XV_S47_1_OpenCommand : BOOL;
   XV_S47_1_Simulation : BOOL;
   XV_S47_2 : AStd_VlvOC;
   XV_S47_2_AOI : AStd_VlvOC_AOI := (cfgHasZSO := 1);
   XV_S47_2_CloseCommand : BOOL;
   XV_S47_2_IOpn : BOOL;
   XV_S47_2_IsClosed : BOOL := 1;
   XV_S47_2_IsOpen : BOOL;
   XV_S47_2_OCls : BOOL;
   XV_S47_2_OpenCommand : BOOL;
   XV_S47_2_Simulation : BOOL;
   XV_S51_1 : AStd_VlvOC := (AutoS := 1, OpenO := 1, OpenI := 1, AutoCtrlS := 1, cfgHasZSC := 1, AutoCtrlC := 1, CycleCountS := 71, Perm.IntlkS := 1, Perm.SafeS := 1, Perm.InterlockInhibitC := 3, Perm.SafetyInhibitC := 3, Perm.InterlockTimers.Timers[2].PRE := 300000, Perm.InterlockTimers.Timers[3].PRE := 300000, MiscAlm.Tmr.PRE := 30000);
   XV_S51_1_AOI : AStd_VlvOC_AOI := (AutoS := 1, OpenS := 1, Open_O := 1, cfgHasZSC := 1);
   XV_S51_1_IOpn : BOOL;
   XV_S51_1_OCls : BOOL;
   XV_S51_1_Simulation : BOOL;
   XV_S51_2 : AStd_VlvOC := (CloseO := 1, ClosedI := 1, cfgHasZSC := 1, CycleCountS := 242, Perm.IntlkS := 1, Perm.SafeS := 1, MiscAlm.InhibitC := 1, MiscAlm.Tmr.PRE := 30000);
   XV_S51_2_AOI : AStd_VlvOC_AOI := (Closed_I := 1, Close_O := 1, cfgHasZSC := 1);
   XV_S51_2_ClsI : BOOL := 1;
   XV_S51_2_IOpn : BOOL;
   XV_S51_2_OCls : BOOL := 1;
   XV_S51_2CloseC : BOOL;
   XV_S51_2OpenC : BOOL;
   XV_S51_3 : AStd_VlvOC := (CloseO := 1, ClosedI := 1, cfgHasZSC := 1, CycleCountS := 188, Perm.IntlkS := 1, Perm.SafeS := 1, MiscAlm.Tmr.PRE := 30000);
   XV_S51_3_AOI : AStd_VlvOC_AOI := (Closed_I := 1, Close_O := 1, cfgHasZSC := 1);
   XV_S51_3_IOpn : BOOL;
   XV_S51_3_OCls : BOOL := 1;
   XV_S51_3CloseC : BOOL;
   XV_S51_3OpenC : BOOL;
   XV_S51_4 : AStd_VlvOC := (AutoS := 1, CloseO := 1, ClosedI := 1, cfgHasZSC := 1, CycleCountS := 105, Perm.IntlkS := 1, Perm.SafeS := 1, MiscAlm.Tmr.PRE := 30000);
   XV_S51_4_AOI : AStd_VlvOC_AOI := (AutoS := 1, Closed_I := 1, Close_O := 1, cfgHasZSC := 1);
   XV_S51_4_IOpn : BOOL;
   XV_S51_4_OCls : BOOL := 1;
   XV_S51_4_Simulation : BOOL;
   XV_S52_1 : AStd_VlvOC := (CloseO := 1, ClosedI := 1, cfgHasZSC := 1, cfgHasZSO := 1, CycleCountS := 22, Perm.IntlkS := 1, Perm.SafeS := 1, Perm.IntSafDisp := 1, MiscAlm.Tmr.PRE := 30000);
   XV_S52_1_AOI : AStd_VlvOC_AOI := (Closed_I := 1, Close_O := 1, cfgHasZSO := 1, cfgHasZSC := 1); {access Read Only}
   XV_S52_1_ClosedI : ALIAS FOR Local:1:I.Data[27].21;
   XV_S52_1_IOpn : BOOL; {access Read Only}
   XV_S52_1_OCls : BOOL := 1; {access Read Only}
   XV_S52_1_OpenC : ALIAS FOR Local:1:O.Data[12].16;
   XV_S52_1_OpenI : ALIAS FOR Local:1:I.Data[27].22;
   XV_S52_2 : AStd_VlvOC := (CloseO := 1, ClosedI := 1, cfgHasZSC := 1, cfgHasZSO := 1, CycleCountS := 22, Perm.IntlkS := 1, Perm.SafeS := 1, MiscAlm.Tmr.PRE := 30000);
   XV_S52_2_AOI : AStd_VlvOC_AOI := (Closed_I := 1, Close_O := 1, cfgHasZSO := 1, cfgHasZSC := 1); {access Read Only}
   XV_S52_2_ClosedI : ALIAS FOR Local:1:I.Data[27].25;
   XV_S52_2_IOpn : BOOL; {access Read Only}
   XV_S52_2_OCls : BOOL := 1; {access Read Only}
   XV_S52_2_OpenC : ALIAS FOR Local:1:O.Data[12].18;
   XV_S52_2_OpenI : ALIAS FOR Local:1:I.Data[27].26;
   XV_TIEBIT : BOOL[64];
   XV_TIETMR : TIMER[64] := ([0].PRE := 1000, [1].PRE := 1000, [1].ACC := 1000, [1].EN := 1, [1].DN := 1, [2].PRE := 1000, [3].PRE := 1000, [3].ACC := 1003, [3].EN := 1, [3].DN := 1, [4].PRE := 1000, [5].PRE := 1000, [5].ACC := 1000, [5].EN := 1, [5].DN := 1, [6].PRE := 1000, [7].PRE := 1000, [7].ACC := 1000, [7].EN := 1, [7].DN := 1, [8].PRE := 1000, [9].PRE := 1000, [9].ACC := 1003, [9].EN := 1, [9].DN := 1, [10].PRE := 1000, [11].PRE := 1000, [11].ACC := 1000, [11].EN := 1, [11].DN := 1, [12].PRE := 2000, [13].PRE := 2000, [13].ACC := 2003, [13].EN := 1, [13].DN := 1, [14].PRE := 1000, [16].PRE := 1000, [16].ACC := 1004, [16].EN := 1, [16].DN := 1, [17].PRE := 1000, [18].PRE := 1000, [18].ACC := 1001, [18].EN := 1, [18].DN := 1, [19].PRE := 1000, [19].ACC := 1003, [19].EN := 1, [19].DN := 1, [20].PRE := 1000, [21].PRE := 1000, [22].PRE := 1000);
   zoldfe4303sf : REAL := 0.0031458;
   zoldfe4304sf : REAL := 0.000202;
   ZSC_3001 : ALIAS FOR Local:3:I.Data.5;
   ZSC_4301 : ALIAS FOR Local:2:I.Data.1;
   ZSC_4302 : ALIAS FOR Local:2:I.Data.3;
   ZSC_4303_03 : BOOL;
   ZSC_4303_04 : BOOL;
   ZSC_4303_05 : BOOL;
   ZSC_4303_1 : ALIAS FOR Local:2:I.Data.7;
   ZSC_4304 : ALIAS FOR Local:2:I.Data.9;
   ZSC_4304_02 : BOOL := 1;
   ZSC_4304_03 : BOOL;
   ZSC_4304_04 : BOOL;
   ZSC_4320_1 : ALIAS FOR Local:1:I.Data[4].3;
   ZSC_4320_2 : ALIAS FOR Local:1:I.Data[4].1;
   ZSC_5201 : ALIAS FOR Local:1:I.Data[27].5;
   ZSC_5202 : ALIAS FOR Local:1:I.Data[27].7;
   ZSC_5301 : ALIAS FOR Local:1:I.Data[27].9;
   ZSC_5302 : ALIAS FOR Local:1:I.Data[27].11;
   ZSC_K400_03 : BOOL;
   ZSC_K400_04 : BOOL;
   ZSO_3001 : ALIAS FOR Local:3:I.Data.4;
   ZSO_4301 : ALIAS FOR Local:2:I.Data.0;
   ZSO_4302 : ALIAS FOR Local:2:I.Data.2;
   ZSO_4303_03 : BOOL;
   ZSO_4303_04 : BOOL;
   ZSO_4303_05 : BOOL := 1;
   ZSO_4303_1 : ALIAS FOR Local:2:I.Data.6;
   ZSO_4304 : ALIAS FOR Local:2:I.Data.8;
   ZSO_4304_02 : BOOL;
   ZSO_4304_03 : BOOL;
   ZSO_4304_04 : BOOL := 1;
   ZSO_4320_1 : ALIAS FOR Local:1:I.Data[4].2;
   ZSO_4320_2 : ALIAS FOR Local:1:I.Data[4].0;
   ZSO_5201 : ALIAS FOR Local:1:I.Data[27].4;
   ZSO_5202 : ALIAS FOR Local:1:I.Data[27].6;
   ZSO_5301 : ALIAS FOR Local:1:I.Data[27].8;
   ZSO_5302 : ALIAS FOR Local:1:I.Data[27].10;
   ZSO_K400_03 : BOOL := 1;
   ZSO_K400_04 : BOOL := 1;
END_VAR

PROGRAM Deviation_Alarms   (* main routine MainRoutine *)

ROUTINE DevAlarms   (* ladder *)
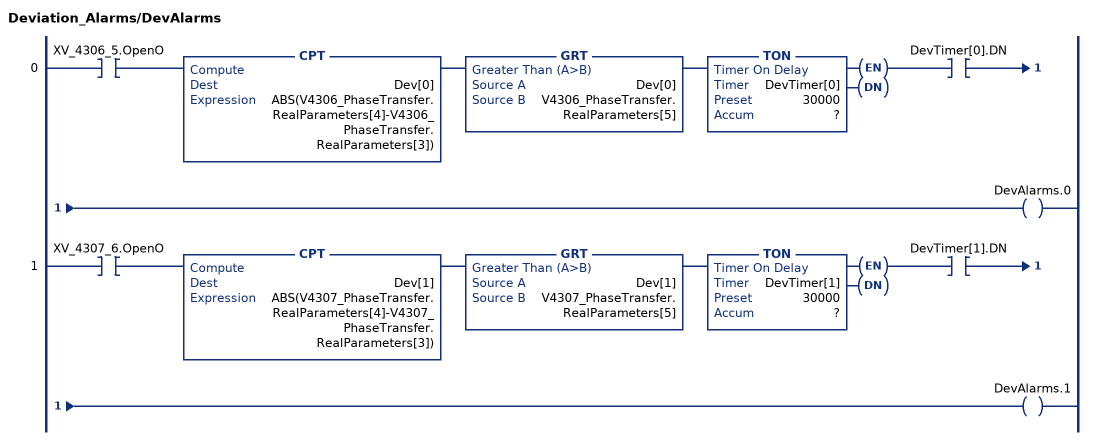
   0: XIC(XV_4306_5.OpenO)CPT(Dev[0],ABS(V4306_PhaseTransfer.RealParameters[4]-V4306_PhaseTransfer.RealParameters[3]))GRT(Dev[0],V4306_PhaseTransfer.RealParameters[5])TON(DevTimer[0],?,?)XIC(DevTimer[0].DN)OTE(DevAlarms.0);
   1: XIC(XV_4307_6.OpenO)CPT(Dev[1],ABS(V4307_PhaseTransfer.RealParameters[4]-V4307_PhaseTransfer.RealParameters[3]))GRT(Dev[1],V4307_PhaseTransfer.RealParameters[5])TON(DevTimer[1],?,?)XIC(DevTimer[1].DN)OTE(DevAlarms.1);
END_ROUTINE

ROUTINE MainRoutine   (* ladder *)
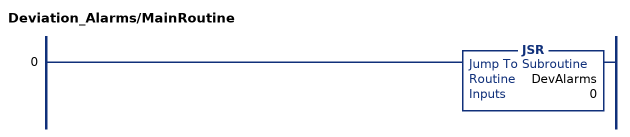
   0: JSR(DevAlarms,0);
END_ROUTINE
END_PROGRAM

PROGRAM General_Purpose   (* main routine MainRoutine *)

ROUTINE GeneralPurpose   (* ladder *)
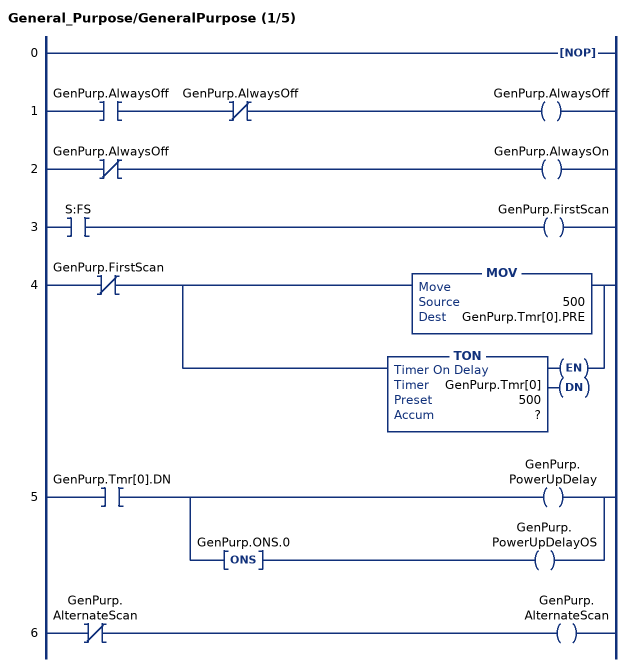
   0: NOP();
   1: XIC(GenPurp.AlwaysOff)XIO(GenPurp.AlwaysOff)OTE(GenPurp.AlwaysOff);
   2: XIO(GenPurp.AlwaysOff)OTE(GenPurp.AlwaysOn);
   3: XIC(S:FS)OTE(GenPurp.FirstScan);
   4: XIO(GenPurp.FirstScan)[MOV(500,GenPurp.Tmr[0].PRE) ,TON(GenPurp.Tmr[0],?,?) ];
   5: XIC(GenPurp.Tmr[0].DN)[OTE(GenPurp.PowerUpDelay) ,ONS(GenPurp.ONS.0) OTE(GenPurp.PowerUpDelayOS) ];
   6: XIO(GenPurp.AlternateScan)OTE(GenPurp.AlternateScan);
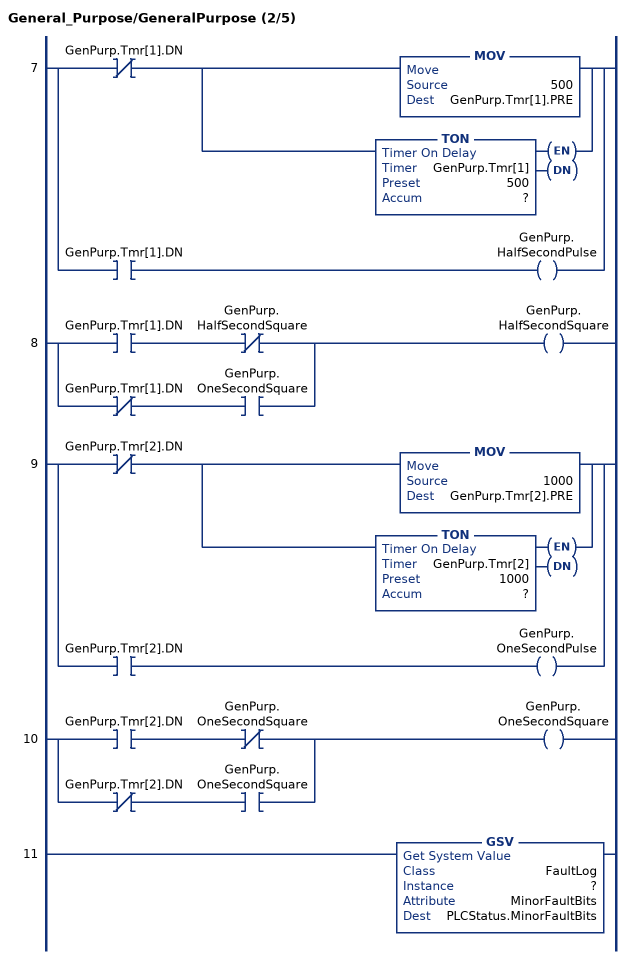
   7: [XIO(GenPurp.Tmr[1].DN) [MOV(500,GenPurp.Tmr[1].PRE) ,TON(GenPurp.Tmr[1],?,?) ] ,XIC(GenPurp.Tmr[1].DN) OTE(GenPurp.HalfSecondPulse) ];
   8: [XIC(GenPurp.Tmr[1].DN) XIO(GenPurp.HalfSecondSquare) ,XIO(GenPurp.Tmr[1].DN) XIC(GenPurp.OneSecondSquare) ]OTE(GenPurp.HalfSecondSquare);
   9: [XIO(GenPurp.Tmr[2].DN) [MOV(1000,GenPurp.Tmr[2].PRE) ,TON(GenPurp.Tmr[2],?,?) ] ,XIC(GenPurp.Tmr[2].DN) OTE(GenPurp.OneSecondPulse) ];
   10: [XIC(GenPurp.Tmr[2].DN) XIO(GenPurp.OneSecondSquare) ,XIO(GenPurp.Tmr[2].DN) XIC(GenPurp.OneSecondSquare) ]OTE(GenPurp.OneSecondSquare);
   11: GSV(FaultLog,?,MinorFaultBits,PLCStatus.MinorFaultBits);
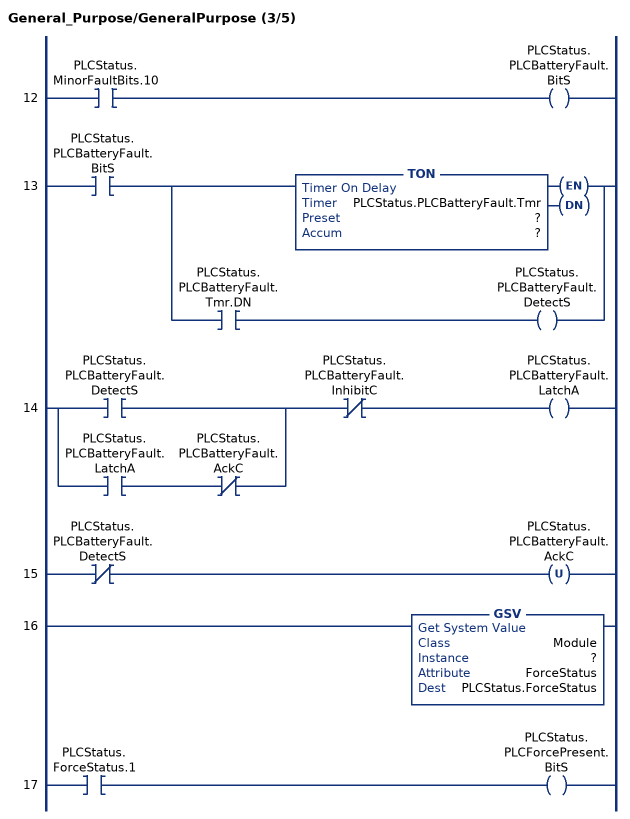
   12: XIC(PLCStatus.MinorFaultBits.10)OTE(PLCStatus.PLCBatteryFault.BitS);
   13: XIC(PLCStatus.PLCBatteryFault.BitS)[TON(PLCStatus.PLCBatteryFault.Tmr,?,?) ,XIC(PLCStatus.PLCBatteryFault.Tmr.DN) OTE(PLCStatus.PLCBatteryFault.DetectS) ];
   14: [XIC(PLCStatus.PLCBatteryFault.DetectS) ,XIC(PLCStatus.PLCBatteryFault.LatchA) XIO(PLCStatus.PLCBatteryFault.AckC) ]XIO(PLCStatus.PLCBatteryFault.InhibitC)OTE(PLCStatus.PLCBatteryFault.LatchA);
   15: XIO(PLCStatus.PLCBatteryFault.DetectS)OTU(PLCStatus.PLCBatteryFault.AckC);
   16: GSV(Module,?,ForceStatus,PLCStatus.ForceStatus);
   17: XIC(PLCStatus.ForceStatus.1)OTE(PLCStatus.PLCForcePresent.BitS);
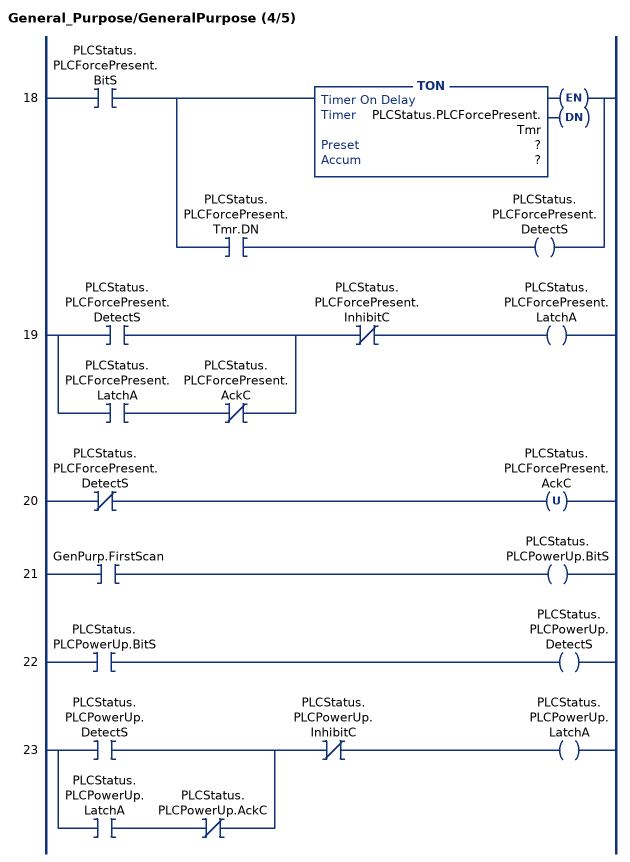
   18: XIC(PLCStatus.PLCForcePresent.BitS)[TON(PLCStatus.PLCForcePresent.Tmr,?,?) ,XIC(PLCStatus.PLCForcePresent.Tmr.DN) OTE(PLCStatus.PLCForcePresent.DetectS) ];
   19: [XIC(PLCStatus.PLCForcePresent.DetectS) ,XIC(PLCStatus.PLCForcePresent.LatchA) XIO(PLCStatus.PLCForcePresent.AckC) ]XIO(PLCStatus.PLCForcePresent.InhibitC)OTE(PLCStatus.PLCForcePresent.LatchA);
   20: XIO(PLCStatus.PLCForcePresent.DetectS)OTU(PLCStatus.PLCForcePresent.AckC);
   21: XIC(GenPurp.FirstScan)OTE(PLCStatus.PLCPowerUp.BitS);
   22: XIC(PLCStatus.PLCPowerUp.BitS)OTE(PLCStatus.PLCPowerUp.DetectS);
   23: [XIC(PLCStatus.PLCPowerUp.DetectS) ,XIC(PLCStatus.PLCPowerUp.LatchA) XIO(PLCStatus.PLCPowerUp.AckC) ]XIO(PLCStatus.PLCPowerUp.InhibitC)OTE(PLCStatus.PLCPowerUp.LatchA);
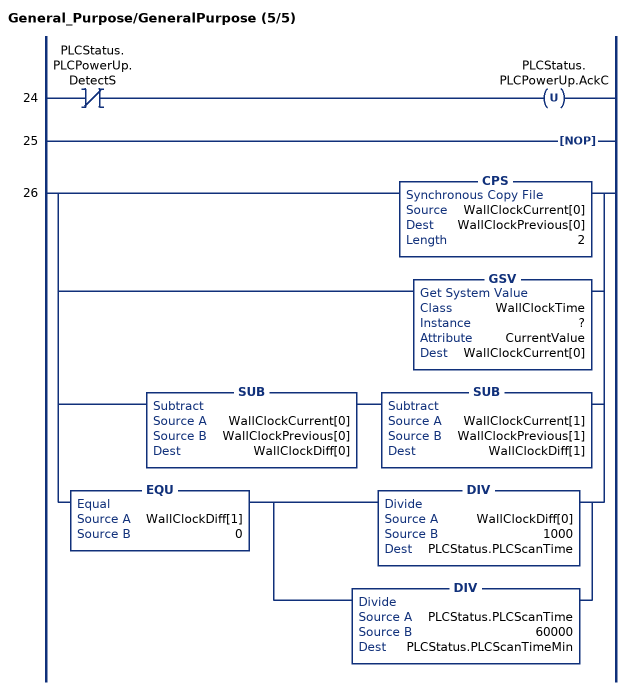
   24: XIO(PLCStatus.PLCPowerUp.DetectS)OTU(PLCStatus.PLCPowerUp.AckC);
   25: NOP();
   26: [CPS(WallClockCurrent[0],WallClockPrevious[0],2) ,GSV(WallClockTime,?,CurrentValue,WallClockCurrent[0]) ,SUB(WallClockCurrent[0],WallClockPrevious[0],WallClockDiff[0]) SUB(WallClockCurrent[1],WallClockPrevious[1],WallClockDiff[1]) ,EQU(WallClockDiff[1],0) [DIV(WallClockDiff[0],1000,PLCStatus.PLCScanTime) ,DIV(PLCStatus.PLCScanTime,60000,PLCStatus.PLCScanTimeMin) ] ];
END_ROUTINE

ROUTINE MainRoutine   (* ladder *)
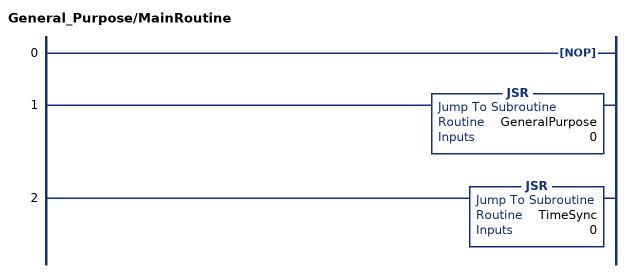
   0: NOP();
   1: JSR(GeneralPurpose,0);
   2: JSR(TimeSync,0);
END_ROUTINE
